(* ========================================================= *)
(*     FB: HLI_CNCChannel                                    *)
(* --------------------------------------------------------- *)
(*   Desc:                                                   *)
(*   Author: MK ,MiB, TV, Rch                                *)
(*   Date: 2020.07.27                                        *)
(*   Rev.: 1.20                                               *)
(*         1.2 Before "start" the state is swicthed to 		 *)
(*				"Selected" and "Ready" to ensure that the    *)	
(*				actual selected program will start 			 *)
(*		   	1.3  BugFix : nChanNo at HLI3_ChannelModeMDI()    *)
(*         	1.4  Implement state switch to "selected" and "ready"  *)         
(*		   	1.5  Channel reset via commanding state 			 *)
(*              RESETTING directly							 *)  
(*		   	1.6  Optimized Channel reset via commanding state *)
(*				RESETTING directly						     *)
(*		   	1.7  Init Paramerer for Manual mode as input parameter*)
(*		   	1.8  BugFix : max index for HLI3_AxisReset		*)
(*		   	1.9  Implementation of HLI3_ManualModeHandler	*)
(*		   	1.10 Implementation of Input bM30Acknowledgement	*)
(*		   	1.12 Optimized Operating modes					*)
(*		   	1.13 Optimized Operating modes				    *)
(*		   	1.14 Optimized M and H Function during Reset     *)
(*		   	1.15 Implementation of ST_CNC_CH_Options Structure *)
(*		   	1.16 BugFix: bCmdReset in mode "Standby" now working *)
(*			1.17 Implementation of CNC PLC Watchdog			*)  
(*			1.18 Optimized CNC PLC Watchdog					*)
(*			1.18 Optimized G201 ManualMode					*)
(*			1.19 Add CmdStandby 							*)
(*			1.20 New Manual Mode 							*)
(* =========================================================*)

IF NOT HLI3_CheckChannelValid(nChannel := nChanIdx) THEN
	RETURN;
END_IF

// CNC PLC Watchdog	
IF NOT stOptions.bDisableCNCPLCWatchDog THEN
	HLI3_SetPLCAlive(nChanIdx :=  nChanIdx);
END_IF

(* handle reset request *)
fbRTrigReset
	(CLK := bStateReset);
	
IF fbRTrigReset.Q THEN
	nStateAutoMDIStart := 0;
	CNCSystem.Channel[nChanIdx].ToolData.bOldToolDataExist := FALSE;
	CNCSystem.Channel[nChanIdx].ToolData.bToolRequest := FALSE;
	CNCSystem.Channel[nChanIdx].ToolData.bResetToolRequest := TRUE;
END_IF

fbRTrigCmdAutomatic(CLK:=bCmdAutomatic);
fbRTrigCmdManual(CLK:=bCmdManual);
fbRTrigCmdReference(CLK:=bCmdReference);
fbRTrigCmdMDI(CLK:=bCmdMDI);
fbRTrigCmdStandby(CLK:=bCmdStandby);	

fbRTrigCmdStart(CLK:=bCmdStart);  
fbRTrigCmdStop(CLK:=bCmdStop);
fbRTrigCmdReset(CLK:=bCmdReset);

(* ************************************* *)
(*  Motion-Control                       *)
(* ************************************* *)

(* EmergencyStop *)
HLI3_ChannelSetEmergencyStop(nChanIdx:=nChanIdx, bEStop := bEmergencyStop);
 
(* Feed Override [0.1%] *)
HLI3_SetChannelOverride(nChanIdx:=nChanIdx, nOverride := nFeedOverride);

(* Rapid feed override [0.1%], must be activated with parameter P-CHAN-00181 *)
HLI3_SetChannelRapidOverride(nChanIdx:=nChanIdx, nOverride := nRapidFeedOverride);

(* Backward Motion *)
HLI3_ChannelSetBackwardMotion(nChanIdx:=nChanIdx, bBackwardMotion:=bBackwardMotion);

(* Program Block Ignore *)
HLI3_ChannelSetProgramBlockIgnore(nChanIdx:=nChanIdx, bPrgBlockIgnore:=bPrgBlockIgnore);

(* Feed Hold *)
HLI3_ChannelSetFeedHold(nChanIdx:=nChanIdx, bFeedHold:=bFeedHold);

(* Single Step *)
HLI3_ChannelSetSingleBlock(nChanIdx:=nChanIdx, bSingleBlock:=bSingleBlock);

(* Reduced Feed *)
HLI3_ChannelSetReducedFeed(nChanIdx:=nChanIdx, bReducedFeed:=bReducedFeed);

(* Syntax Check *)
gpCh[nChanIdx]^.decoder_mc_control.execution_mode.command_w := nSyntaxCheck;

(* Optional stop M01 *)
gpCh[nChanIdx]^.bahn_mc_control.m01_stop_enable.command_w := bM01Stop;

(* ************************************ *)
(*  MHT-Function                        *)
(* ************************************ *)

(* MHT-Function, channel *)
IF NOT stOptions.bDisableMFunctHandling THEN
	ChannelMHTFunction(nChanIdx:=nChanIdx, bM30Acknowledgement := bM30Acknowledgement);
END_IF

(* ************************************* *)
(*  Channel Status Info and error        *)
(* ************************************* *)
HLI3_GetChannelStatusInfo(nChanIdx:=nChanIdx);
HLI3_GetChannelError(nChanIdx:=nChanIdx);

(* ************************************* *)
(*  do single stepping                   *)
(* ************************************* *)
(* Achtung: hier noch anpassen, nur in Abhaengigkeit vom aktuellen Status den Start setzen *)
IF bDoSingleBlock THEN
	bDoSingleBlock := FALSE;
	bStateStart 	:= TRUE;
END_IF

(* ************************************* *)
(*  Operation Modes                      *)
(* ************************************* *)
(* Target modes and states *)
pChannel := ADR(CNCSystem.Channel[nChanIdx]);
OpModes();

(* OperationMode Standby *)
IF stCmdModesStates.stModes.Standby = TRUE THEN
	HLI3_ChannelModeStandby(nChanIdx := nChanIdx,ProgramName:=sProgramName, stCmdModesStates:=stCmdModesStates);
END_IF

(* OperationMode Auto *)
IF stCmdModesStates.stModes.Auto = TRUE THEN
	HLI3_ChannelModeAuto(nChanIdx := nChanIdx, ProgramName:=sProgramName, stCmdModesStates:=stCmdModesStates );
END_IF

(* OperationMode MDI *)
IF stCmdModesStates.stModes.MDI THEN
	(*sProgramName := PLCCncMDIString;*)
	HLI3_ChannelModeMDI(nChanIdx := nChanIdx, pMDIString:=ADR(sMDIString),stCmdModesStates:=stCmdModesStates);
END_IF

(* OperationMode Reference *)
IF stCmdModesStates.stModes.Homing THEN
	sProgramName := '';	(* we choose the default program: rpf.nc *)
	HLI3_ChannelModeReference(nChanIdx := nChanIdx, sRefPosString:=sProgramName, stCmdModesStates:=stCmdModesStates);
END_IF

(* OperationMode Manual *)
(*
IF stCmdModesStates.stModes.Manual THEN	
	HLI3_ChannelModeManual(nChanIdx := nChanIdx, stCmdModesStates:=stCmdModesStates);
END_IF
*)

ModeManual
	(stManualModeParameter  	 	 := stManualModeParameter,
	 stManualModeControlElements	 := stManualModeControlElements,
	 stManualModeControlElementState := stManualModeControlElementState,
	 stCmdModesStates				 := stCmdModesStates,  	
	 arrAxisInG201 				      => stManualModeState[nChanIdx].arrAxisInG201
);
			
(* Reset *)
HLI3_ChannelReset(nChanIdx:=nChanIdx);							(* channel *)
FOR idx := 0 TO UDINT_TO_INT(gNrAx-1) DO							(* axis *)
	HLI3_AxisReset(nChanNo:=nChanIdx+1, nHliAxisIdx:=idx);
END_FOR

ACTION AutoMDIStart:



CASE nStateAutoMDIStart OF
	0:		;(* IDLE *)
	
	10: (* swicth to selected *)
		stCmdModesStates.stStates.Selected := TRUE;
		nStateAutoMDIStart := nStateAutoMDIStart +10;
		
	20: (* wait for selected *)
		IF (pChannel^.ActState =  HLI_IMCM_PROCESS_SELECTED) THEN
			stCmdModesStates.stStates.Ready := TRUE;
			nStateAutoMDIStart := nStateAutoMDIStart +10;
		END_IF
	30: (* Wait for ready and then start*)
		IF (pChannel^.ActState =  HLI_IMCM_PROCESS_READY) THEN
			stCmdModesStates.stStates.Active := TRUE; 
			nStateAutoMDIStart := 0;
		END_IF
	
END_CASE
END_ACTION

ACTION OpModes:
(*************************************************)
(* Restore internal state at first run           *)
(* after PLC reset                               *)
(*************************************************)

IF bCheckOpModeFirst = FALSE THEN
	bCheckOpModeFirst := TRUE;
	currentMode := HLI3_GetChannelMode(nChanIdx:=nChanIdx);
	IF currentMode = HLI_IMCM_STANDBY_MODE THEN
		stCmdModesStates.stModes.Standby := TRUE;
	END_IF
	IF currentMode = HLI_IMCM_AUTOMATIC_MODE THEN
		stCmdModesStates.stModes.Auto := TRUE;
	END_IF
	IF currentMode = HLI_IMCM_MDI_MODE THEN
		stCmdModesStates.stModes.MDI := TRUE;
	END_IF
	IF currentMode = HLI_IMCM_MANUAL_MODE THEN
		stCmdModesStates.stModes.Manual := TRUE;
	END_IF
	IF currentMode = HLI_IMCM_REFERENCE_MODE THEN		
		stCmdModesStates.stModes.Homing := TRUE;
	END_IF
END_IF


(*************************************************)
(* Operation Modes                               *)
(*************************************************)

IF bModeStandby OR fbRTrigCmdStandby.Q THEN
	bModeStandby := FALSE;
	stCmdModesStates.stModes.Standby		:= TRUE;
	stCmdModesStates.stModes.Auto			:= FALSE;
	stCmdModesStates.stModes.MDI			:= FALSE;
	stCmdModesStates.stModes.Manual		:= FALSE;
	stCmdModesStates.stModes.Homing		:= FALSE;
	stCmdModesStates.stStates.Selected	:= TRUE;
END_IF

IF bModeAutomatic OR fbRTrigCmdAutomatic.Q THEN
	bModeAutomatic 				:= FALSE;
	bGoToActive					:= FALSE;
	stCmdModesStates.stModes.Standby		:= FALSE;
	stCmdModesStates.stModes.Auto			:= TRUE;
	stCmdModesStates.stModes.MDI			:= FALSE;
	stCmdModesStates.stModes.Manual		:= FALSE;
	stCmdModesStates.stModes.Homing		:= FALSE;

	stCmdModesStates.stStates.Selected	:= TRUE;
END_IF

IF bModeMDI OR fbRTrigCmdMDI.Q THEN
	bModeMDI := FALSE;
	bGoToActive					:= FALSE;
	stCmdModesStates.stModes.Standby		:= FALSE;
	stCmdModesStates.stModes.Auto			:= FALSE;
	stCmdModesStates.stModes.MDI			:= TRUE;
	stCmdModesStates.stModes.Manual		:= FALSE;
	stCmdModesStates.stModes.Homing		:= FALSE;

	stCmdModesStates.stStates.Selected	:= TRUE;
END_IF

IF bModeManual OR fbRTrigCmdManual.Q THEN
	bModeManual := FALSE;
	stCmdModesStates.stModes.Standby		:= FALSE;
	stCmdModesStates.stModes.Auto			:= FALSE;
	stCmdModesStates.stModes.MDI			:= FALSE;
	stCmdModesStates.stModes.Manual		:= TRUE;
	stCmdModesStates.stModes.Homing		:= FALSE;

	stCmdModesStates.stStates.Active		:= TRUE;
END_IF

IF bModeReference OR fbRTrigCmdReference.Q THEN
	bModeReference := FALSE;
	bGoToActive					:= FALSE;
	stCmdModesStates.stModes.Standby		:= FALSE;
	stCmdModesStates.stModes.Auto			:= FALSE;
	stCmdModesStates.stModes.MDI			:= FALSE;
	stCmdModesStates.stModes.Manual		:= FALSE;
	stCmdModesStates.stModes.Homing		:= TRUE;
	
	IF stOptions.bReferenceModeStartRequired THEN
		stCmdModesStates.stStates.Selected	:= TRUE;
	ELSE
		stCmdModesStates.stStates.Active	:= TRUE;			
	END_IF	
	
END_IF



(*************************************************)
(* Operation States                              *)
(*************************************************)

currentMode := HLI3_GetChannelMode(nChanIdx:=nChanIdx);
currentState := HLI3_GetChannelState(nChanIdx:=nChanIdx);

CASE currentMode OF
	(*-------------------------------------------------------------------*)
	HLI_IMCM_STANDBY_MODE:
		IF bStateReset OR fbRTrigCmdReset.Q THEN
			stCmdModesStates.stModes.Standby := TRUE;
			stCmdModesStates.stStates.Reset := TRUE;
			CNCSystem.Channel[nChanIdx].ToolData.bOldToolDataExist := FALSE;
			CNCSystem.Channel[nChanIdx].ToolData.bToolRequest := FALSE;
			CNCSystem.Channel[nChanIdx].ToolData.bResetToolRequest := TRUE;		
		END_IF

	(*-------------------------------------------------------------------*)
	HLI_IMCM_AUTOMATIC_MODE:
		IF bStateStart OR fbRTrigCmdStart.Q THEN  (* replaced a simple 'start' by a sequence which switches the state to selected and ready*)
			IF currentState <> HLI_IMCM_PROCESS_HOLD AND currentState <> HLI_IMCM_PROCESS_ACTIVE THEN
				nStateAutoMDIStart := 10;
			ELSE
				stCmdModesStates.stStates.Active := TRUE; 
			END_IF					   	
		END_IF
		IF nStateAutoMDIStart <> 0 THEN
			AutoMDIStart();
		END_IF

		IF (bStateStop OR fbRTrigCmdStop.Q) AND currentState <> HLI_IMCM_PROCESS_DESELECTED THEN
			stCmdModesStates.stStates.Hold := TRUE;
		END_IF

		IF bStateReady THEN
			stCmdModesStates.stStates.Ready := TRUE;
		END_IF

		IF bStateReset OR fbRTrigCmdReset.Q THEN
			stCmdModesStates.stStates.Reset := TRUE;
			CNCSystem.Channel[nChanIdx].ToolData.bOldToolDataExist := FALSE;
			CNCSystem.Channel[nChanIdx].ToolData.bToolRequest := FALSE;
			CNCSystem.Channel[nChanIdx].ToolData.bResetToolRequest := TRUE;			
		END_IF
		
		IF bStateSelect THEN
			stCmdModesStates.stStates.Selected := TRUE;
		END_IF		

	(*-------------------------------------------------------------------*)
	HLI_IMCM_MDI_MODE:
		IF bStateStart OR fbRTrigCmdStart.Q THEN
			IF currentState <> HLI_IMCM_PROCESS_HOLD AND currentState <> HLI_IMCM_PROCESS_ACTIVE THEN
				nStateAutoMDIStart := 10;
			ELSE
				stCmdModesStates.stStates.Active := TRUE; 
			END_IF
		END_IF
		
		IF nStateAutoMDIStart <> 0 THEN
			AutoMDIStart();
		END_IF
		
		IF (bStateStop OR fbRTrigCmdStop.Q) AND currentState <> HLI_IMCM_PROCESS_DESELECTED THEN
			stCmdModesStates.stStates.Hold := TRUE;
		END_IF

		IF bStateSelect THEN
			stCmdModesStates.stStates.Selected := TRUE;
		END_IF
		
		IF bStateReady THEN
			stCmdModesStates.stStates.Ready := TRUE;
		END_IF

		IF bStateReset OR fbRTrigCmdReset.Q THEN
			stCmdModesStates.stStates.Reset := TRUE;
			CNCSystem.Channel[nChanIdx].ToolData.bOldToolDataExist := FALSE;
			CNCSystem.Channel[nChanIdx].ToolData.bToolRequest := FALSE;
			CNCSystem.Channel[nChanIdx].ToolData.bResetToolRequest := TRUE;			
		END_IF

	(*-------------------------------------------------------------------*)
	HLI_IMCM_MANUAL_MODE:
		IF bStateStart OR fbRTrigCmdStart.Q OR ((currentState = HLI_IMCM_PROCESS_SELECTED) AND bGoToActive) THEN
			bGoToActive := FALSE;	
			stCmdModesStates.stStates.Active 	:= TRUE;
		END_IF

		IF bStateReady THEN
			stCmdModesStates.stStates.Ready 	:= TRUE;
		END_IF

		IF bStateSelect THEN
			stCmdModesStates.stStates.Selected := TRUE;
		END_IF

		IF bStateStop OR fbRTrigCmdStop.Q THEN
			stCmdModesStates.stStates.Hold := TRUE;
		END_IF

		IF (bStateReset OR fbRTrigCmdReset.Q) THEN	
			CNCSystem.Channel[nChanIdx].ToolData.bOldToolDataExist := FALSE;
			CNCSystem.Channel[nChanIdx].ToolData.bToolRequest := FALSE;
			CNCSystem.Channel[nChanIdx].ToolData.bResetToolRequest := TRUE;
			
			stCmdModesStates.stStates.Reset := TRUE;
			IF stCmdModesStates.stModes.Manual THEN
				bGoToActive := TRUE;
			END_IF
		END_IF

	(*-------------------------------------------------------------------*)
	HLI_IMCM_REFERENCE_MODE:
		IF bStateStart OR fbRTrigCmdStart.Q THEN
			stCmdModesStates.stStates.Active := TRUE;
		END_IF

		IF bStateStop OR fbRTrigCmdStop.Q THEN
			stCmdModesStates.stStates.Hold := TRUE;
		END_IF

		IF bStateReset OR fbRTrigCmdReset.Q THEN
			CNCSystem.Channel[nChanIdx].ToolData.bOldToolDataExist := FALSE;
			CNCSystem.Channel[nChanIdx].ToolData.bToolRequest := FALSE;
			CNCSystem.Channel[nChanIdx].ToolData.bResetToolRequest := TRUE;			
			stCmdModesStates.stStates.Reset := TRUE;
		END_IF
END_CASE


bStateStart 	:= FALSE;
bStateStop 		:= FALSE;
bStateReset 	:= FALSE;
bStateSelect 	:= FALSE;
bStateready 	:= FALSE;
END_ACTION

END_FUNCTION_BLOCK

// CNC/8 Mis/HLI3_SetPLCAlive
FUNCTION HLI3_SetPLCAlive : BOOL
VAR_INPUT
	nChanIdx: INT;		
END_VAR

VAR
	nWatchdogCycles 	: UDINT :=2;	 	
END_VAR

(*
Display PLC is just alive (Trigger Watchdog to MC)
If PLC is stopped here, alive sign is missing.
-> CNC raises error message
-> CNC stoppes movement with internal FEEDHOLD
-> system has to be restarted (after removal of error)
*)

HLI3_SetPLCAlive := FALSE;
IF NOT HLI3_CheckChannelValid(nChannel := nChanIdx) THEN
	RETURN;
END_IF

nWatchdogCycles := 2;

gpCh[nChanIdx]^.head.mc_watchdog.cycle_time_w := CNCSystem.nPLCCycleTime * nWatchdogCycles;   // Watchdog time : PLC Cycle Time * nWatchdogCycles
gpCh[nChanIdx]^.head.mc_watchdog.enable_w := TRUE;
gpCh[nChanIdx]^.head.mc_watchdog.alive_rw := TRUE;

HLI3_SetPLCAlive := TRUE;

END_FUNCTION

// CNC/3 Control/HLI3_ChannelSetEmergencyStop
FUNCTION HLI3_ChannelSetEmergencyStop : BOOL
VAR_INPUT
	/// Number of channel 
	nChanIdx: INT;
	bEStop: BOOL;
END_VAR

(****************************************************************************************)
(* POU:			HLI_ChannelSetEmergenyStop												*)
(* Type:		Function block															*)
(* Customer:	Common																	*)
(* Date:		09/03/12																*)
(* Last:		20/11/12																*)
(* ------------------------------------------------------------------------------------ *)
(* Revision:	1.0																		*)
(* Author:		HR,MiB																	*)
(* Description: (Re-)Sets the channel specific emergency stop unit.						*)
(****************************************************************************************)

HLI3_ChannelSetEmergencyStop := FALSE;
IF NOT HLI3_CheckChannelValid(nChannel := nChanIdx) THEN
	RETURN;
END_IF

(* if the stop button from the HMI is selected the request is set *)
gpCh[nChanIdx]^.bahn_mc_control.emergency_stop.command_w := bEStop;

HLI3_ChannelSetEmergencyStop		:= TRUE;

END_FUNCTION

// CNC/3 Control/HLI3_SetChannelOverride
FUNCTION HLI3_SetChannelOverride : BOOL
VAR_INPUT
	/// Number of channel 
	nChanIdx: INT;
	nOverride: UINT;
END_VAR

(* ========================================================= *)
(*    FUN: HLI_SetChannelOverride                            *)
(* --------------------------------------------------------- *)
(*   Desc: Set the channel Override                          *)
(* Author: MK, MiB                                           *)
(*   Date: 20.11.2012                                        *)
(*   Rev.: 1.2  2017.10.25                                   *)
(* ========================================================= *)

IF NOT HLI3_CheckChannelValid(nChannel := nChanIdx) THEN
	HLI3_SetChannelOverride := FALSE;
	RETURN;
END_IF

(* Limit the override *)
IF nOverride > 2000 THEN nOverride := 2000; END_IF  // MiB 2017.10.25 valid maximum in cnc core is 2000
IF nOverride < 0 THEN nOverride := 0; END_IF

gpCh[nChanIdx]^.bahn_mc_control.override_feedrate.command_w := nOverride;

HLI3_SetChannelOverride := TRUE;

END_FUNCTION

// CNC/3 Control/HLI3_SetChannelRapidOverride
FUNCTION HLI3_SetChannelRapidOverride : BOOL
VAR_INPUT
	/// Number of channel 
	nChanIdx: INT;
	nOverride: UINT;
END_VAR

(* ========================================================= *)
(*    FUN: HLI_SetChannelRapidOverride                       *)
(* --------------------------------------------------------- *)
(*   Desc: Set the channel Override for rapid movements      *)
(*   Author: TV , MiB                                        *)
(*   Date: 07.02.2017                                        *)
(*   Rev.: 1.1                                               *)
(* ========================================================= *)

IF NOT HLI3_CheckChannelValid(nChannel := nChanIdx) THEN
	HLI3_SetChannelRapidOverride := FALSE;
	RETURN;
END_IF

(* Limit the override *)
IF nOverride > 1000	THEN nOverride := 1000; END_IF  // MiB 2017.10.25 maximum is 1000 (ref HLI manual)
IF nOverride < 0 THEN nOverride := 0; END_IF

gpCh[nChanIdx]^.bahn_mc_control.override_rapid_move.enable_w := TRUE;
gpCh[nChanIdx]^.bahn_mc_control.override_rapid_move.command_w := nOverride;

HLI3_SetChannelRapidOverride := TRUE;

END_FUNCTION

// CNC/3 Control/HLI3_ChannelSetBackwardMotion
FUNCTION HLI3_ChannelSetBackwardMotion : BOOL
VAR_INPUT
	/// Number of channel 
	nChanIdx: INT;
	bBackwardMotion: BOOL;
END_VAR

(* ========================================================= *)
(*    FUN: HLI_ChannelSetBackwardMotion                      *)
(* --------------------------------------------------------- *)
(*   Desc:                                                   *)
(* Author: MK, MiB                                           *)
(*   Date: 20.11.2012                                        *)
(*   Rev.: 1.1                                               *)
(* ========================================================= *)

HLI3_ChannelSetBackwardMotion := FALSE;
IF NOT HLI3_CheckChannelValid(nChannel := nChanIdx) THEN
	RETURN;
END_IF

gpCh[nChanIdx]^.bahn_mc_control.backward_motion.command_w := bBackwardMotion;

HLI3_ChannelSetBackwardMotion := TRUE;

END_FUNCTION

// CNC/3 Control/HLI3_ChannelSetProgramBlockIgnore
FUNCTION HLI3_ChannelSetProgramBlockIgnore : BOOL
VAR_INPUT
	/// Number of channel 
	nChanIdx: INT;
	bPrgBlockIgnore: BOOL;
END_VAR

(* ========================================================= *)
(*    FUN: HLI_SetProgramBlockIgnore                         *)
(* --------------------------------------------------------- *)
(*   Desc:                                                   *)
(* Author: MK, MiB , TV                                      *)
(*   Date: 20.12.2012                                        *)
(*   Last: 19.11.2013                                        *)
(*   Rev.: 1.0                                               *)
(* ========================================================= *)

HLI3_ChannelSetProgramBlockIgnore := FALSE;
IF NOT HLI3_CheckChannelValid(nChannel := nChanIdx) THEN
	RETURN;
END_IF

(* program block ignore *)
IF bPrgBlockIgnore THEN
	gpCh[nChanIdx]^.decoder_mc_control.program_block_ignore.command_w := 1;
ELSE
	gpCh[nChanIdx]^.decoder_mc_control.program_block_ignore.command_w := 0;
END_IF

HLI3_ChannelSetProgramBlockIgnore := TRUE;

END_FUNCTION

// CNC/3 Control/HLI3_ChannelSetFeedHold
FUNCTION HLI3_ChannelSetFeedHold : BOOL
VAR_INPUT
	/// Number of channel 
	nChanIdx: INT;
	bFeedHold: BOOL;
END_VAR

(* ========================================================= *)
(*    FUN: HLI_ChannelSetFeedHold                            *)
(* --------------------------------------------------------- *)
(*   Desc:                                                   *)
(* Author: MK , MiB                                          *)
(*   Date: 20.11.2012                                        *)
(*   Rev.: 1.1                                               *)
(* ========================================================= *)

HLI3_ChannelSetFeedHold := FALSE;
IF NOT HLI3_CheckChannelValid(nChannel := nChanIdx) THEN
	RETURN;
END_IF

(* if the stop button from the HMI is selected the request is set *)
gpCh[nChanIdx]^.bahn_mc_control.feedhold.command_w := bFeedHold OR gpCh[nChanIdx]^.bahn_mc_control.feedhold.request_r;
HLI3_ChannelSetFeedHold := TRUE;

END_FUNCTION

// CNC/3 Control/HLI3_ChannelSetSingleBlock
FUNCTION HLI3_ChannelSetSingleBlock : BOOL
VAR_INPUT
	/// Number of channel 
	nChanIdx: INT;
	bSingleBlock: BOOL;
END_VAR

(* ========================================================= *)
(*    FUN: HLI3_ChannelSetSingleBlock                        *)
(* --------------------------------------------------------- *)
(*   Desc:                                                   *)
(* Author: MK ,MiB                                           *)
(*   Date: 20.11.2012                                        *)
(*   Rev.: 1.1                                               *)
(* ========================================================= *)

HLI3_ChannelSetSingleBlock := FALSE;
IF NOT HLI3_CheckChannelValid(nChannel := nChanIdx) THEN
	RETURN;
END_IF
gpCh[nChanIdx]^.bahn_mc_control.single_block.command_w   := bSingleBlock;

HLI3_ChannelSetSingleBlock := TRUE;

END_FUNCTION

// CNC/3 Control/HLI3_ChannelSetReducedFeed
FUNCTION HLI3_ChannelSetReducedFeed : BOOL
VAR_INPUT
	/// Number of channel 
	nChanIdx: INT;
	bReducedFeed: BOOL;
END_VAR

(* ========================================================= *)
(*    FUN: HLI_ChannelSetReducedFeed                         *)
(* --------------------------------------------------------- *)
(*   Desc:                                                   *)
(* Author: MK,MiB                                            *)
(*   Date: 20.11.2012                                        *)
(*   Rev.: 1.1                                               *)
(* ========================================================= *)


HLI3_ChannelSetReducedFeed := FALSE;
IF NOT HLI3_CheckChannelValid(nChannel := nChanIdx) THEN
	RETURN;
END_IF
gpCh[nChanIdx]^.bahn_mc_control.reduced_speed.command_w := bReducedFeed;
HLI3_ChannelSetReducedFeed := TRUE;

END_FUNCTION

// CNC/3 Control/HLI3_GetChannelStatusInfo
FUNCTION HLI3_GetChannelStatusInfo : BOOL
VAR_INPUT
	/// Number of channel 
	nChanIdx: INT;
END_VAR
VAR
	pChannel: POINTER TO ST_CNCChannel;
END_VAR

(* ========================================================= *)
(*    FUN: HLI_GetStatusInfo                                 *)
(* --------------------------------------------------------- *)
(*   Desc: Status Info from the HLI Interface                *)
(* Author: MK,Mib                                            *)
(*   Date: 18.07.2002                                        *)
(*   Rev.: 1.0                                               *)
(* ========================================================= *)

IF NOT HLI3_CheckChannelValid(nChannel := nChanIdx) THEN
	RETURN;
END_IF


pChannel := ADR(CNCSystem.Channel[nChanIdx]);
pChannel^.ActMode := HLI3_GetChannelMode(nChanIdx:=nChanIdx);
pChannel^.ActState := HLI3_GetChannelState(nChanIdx:=nChanIdx);

pChannel^.Mode.Standby := FALSE;
pChannel^.Mode.Auto := FALSE;
pChannel^.Mode.Homing := FALSE;
pChannel^.Mode.MDI := FALSE;
pChannel^.Mode.Manual := FALSE;

(* Translate mode *)
CASE pChannel^.ActMode OF
	HLI_IMCM_MODE:					pChannel^.ActModeString := 'Mode';
	HLI_IMCM_STANDBY_MODE:			pChannel^.ActModeString := 'StandbyMode'; pChannel^.Mode.Standby:=TRUE;
	HLI_IMCM_AUTOMATIC_MODE:		pChannel^.ActModeString := 'AutomaticMode'; pChannel^.Mode.Auto:=TRUE;
	HLI_IMCM_MDI_MODE:				pChannel^.ActModeString := 'MDIMode'; pChannel^.Mode.MDI:=TRUE;
	HLI_IMCM_MANUAL_MODE:			pChannel^.ActModeString := 'ManualMode'; pChannel^.Mode.Manual:=TRUE;;
	HLI_IMCM_REFERENCE_MODE:		pChannel^.ActModeString := 'ReferenceMode'; pChannel^.Mode.Homing:=TRUE;
ELSE
	pChannel^.ActModeString := '---';
END_CASE;

pChannel^.State.Selected:=FALSE;
pChannel^.State.Ready:=FALSE;
pChannel^.State.Active:=FALSE;
pChannel^.State.Hold:=FALSE;
pChannel^.State.Error:=FALSE;

(* Translate state *)
CASE pChannel^.ActState OF
	HLI_IMCM_PROCESS_DESELECTED:	pChannel^.ActStateString := 'Deselected';
	HLI_IMCM_PROCESS_SELECTED:		pChannel^.ActStateString := 'Selected'; pChannel^.State.Selected:=TRUE;
	HLI_IMCM_PROCESS_READY:			pChannel^.ActStateString := 'Ready'; pChannel^.State.Ready:=TRUE;
	HLI_IMCM_PROCESS_ACTIVE:		pChannel^.ActStateString := 'Active'; pChannel^.State.Active:=TRUE;
	HLI_IMCM_PROCESS_HOLD:			pChannel^.ActStateString := 'Hold'; pChannel^.State.Hold:=TRUE;
	HLI_IMCM_PROCESS_ERROR:			pChannel^.ActStateString := 'Error'; pChannel^.State.Error:=TRUE;
	HLI_IMCM_PROCESS_SELECTING:		pChannel^.ActStateString := 'Selecting';
	HLI_IMCM_PROCESS_DESELECTING:	pChannel^.ActStateString := 'Deselecting';
	HLI_IMCM_PROCESS_PREPARING:		pChannel^.ActStateString := 'Preparing';
	HLI_IMCM_PROCESS_CLEARING:		pChannel^.ActStateString := 'Clearing';
	HLI_IMCM_PROCESS_STARTING:		pChannel^.ActStateString := 'Starting';
	HLI_IMCM_PROCESS_ABORTING:		pChannel^.ActStateString := 'Aborting';
	HLI_IMCM_PROCESS_STOPPING:		pChannel^.ActStateString := 'Stopping';
	HLI_IMCM_PROCESS_RESUMING:		pChannel^.ActStateString := 'Resuming';
	HLI_IMCM_PROCESS_RESETTING:		pChannel^.ActStateString := 'Resetting';
	HLI_IMCM_PROCESS_FINISHING:		pChannel^.ActStateString := 'Finishing';
ELSE
	pChannel^.ActStateString := '---';
END_CASE;

END_FUNCTION

// CNC/3 Control/HLI3_GetChannelMode
FUNCTION HLI3_GetChannelMode : UDINT
VAR_INPUT
	/// Number of channel 
	nChanIdx: INT;
END_VAR

(* ========================================================= *)
(*    FUN: HLI_GetChannelMode                                *)
(* --------------------------------------------------------- *)
(*   Desc:                                                   *)
(* Author: MK                                                *)
(*   Date: 18.07.2002                                        *)
(*   Rev.: 1.0                                               *)
(* ========================================================= *)
HLI3_GetChannelMode := 0;
IF NOT HLI3_CheckChannelValid(nChannel := nChanIdx) THEN
	RETURN;
END_IF

(* if the stop button from the HMI is selected the request is set *)
HLI3_GetChannelMode := gpCh[nChanIdx]^.channel_mc_control.mode_and_state.state_r.mode;

END_FUNCTION

// CNC/3 Control/HLI3_GetChannelState
FUNCTION HLI3_GetChannelState : UDINT
VAR_INPUT
	/// Number of channel 
	nChanIdx: INT;
END_VAR

(* ========================================================= *)
(*    FUN: HLI3_GetChannelState                              *)
(* --------------------------------------------------------- *)
(*   Desc:                                                   *)
(* Author: MK                                                *)
(*   Date: 18.07.2002                                        *)
(*   Rev.: 1.0                                               *)
(* ========================================================= *)

HLI3_GetChannelState := 0;
IF NOT HLI3_CheckChannelValid(nChannel := nChanIdx) THEN
	RETURN;
END_IF

(* if the stop button from the HMI is selected the request is set *)
HLI3_GetChannelState := gpCh[nChanIdx]^.channel_mc_control.mode_and_state.state_r.state;

END_FUNCTION

// CNC/3 Control/HLI3_GetChannelError
FUNCTION HLI3_GetChannelError : BOOL
VAR_INPUT
	/// Number of channel 
	nChanIdx: INT;
END_VAR
VAR
	pChannel: POINTER TO ST_CNCChannel;
END_VAR

(* ========================================================= *)
(*    FUN: HLI_GetChannelError                               *)
(* --------------------------------------------------------- *)
(*   Desc: Gets the channel error                            *)
(* Return: The error flag of the channel                     *)
(* Author: MK , MiB, TV                                      *)
(*   Date: 08.07.2015                                        *)
(*   Rev.: 1.3                                               *)
(* ========================================================= *)

IF NOT HLI3_CheckChannelValid(nChannel := nChanIdx) THEN
	RETURN;
END_IF

pChannel := ADR(CNCSystem.Channel[nChanIdx]);

(* Visualisation of Mode and State *)
pChannel^.ActMode  := HLI3_GetChannelMode(nChanIdx:=nChanIdx);
pChannel^.ActState := HLI3_GetChannelState(nChanIdx:=nChanIdx);

(* Error messages id *)
IF pChannel^.ActState = HLI_IMCM_PROCESS_ERROR THEN
	pChannel^.Error := TRUE;	
ELSE
	pChannel^.Error := FALSE;	
END_IF

END_FUNCTION

// CNC/4 MHT-Function/HLI3_QuitChannelMHTFunction
FUNCTION_BLOCK HLI3_QuitChannelMHTFunction
VAR_INPUT
	/// Number of channel 
	nChanIdx: INT;
	bM30Acknowledgement : BOOL;
END_VAR
VAR_OUTPUT
	bOK: BOOL;
END_VAR
VAR
	ChannelMFunction: HLI3_DoChannelMFunction;
	ChannelTFunction: HLI3_DoChannelTFunction;
	ChannelHFunction: HLI3_DoChannelHFunction;
	/// local pointer to Data of actual Channel 
	pChannelData: POINTER TO HIGH_LEVEL_INTERFACE_CH;
	/// local pointer to actual techno unit 
	pActTechnoUnit: POINTER TO TECHNO_UNIT_CH;
	/// Index of axis specific technology function at HLI 
	nTechFctMaxIdx: UINT;
	nTechFctAnzahl : UINT; 
	/// loop variable 
	idx: UINT;
	/// number of M-function 
	nFuncNr: UDINT;
	nArgument: DINT;
	/// basis id of a tool 
	nToolBasicId: UDINT;
	pMHProcess: POINTER TO HLI_M_H_PROZESS;
	pSProcess: POINTER TO HLI_S_PROZESS;
	pTProcess: POINTER TO HLI_T_PROZESS;
	stAttributeData: St_TechnoAttributeData;	
END_VAR

(* ========================================================= *)
(*     FB: HLI3_QuitChannelMHTFunction                        *)
(* --------------------------------------------------------- *)
(*   Desc:                                                   *)
(* Author: MK                                                *)
(*   Rev.: 1.1                                               *)
(*   Date: 18.07.2002                                        *)
(*       : 08.04.2005                                        *)
(*          24.11.2010 MiB Erweiterung um H Funktionen 		 *)
(* ========================================================= *)
(* Rev.:	1.2												 *)
(* Date:	02.10.2010                                    	 *)
(* Author:	HR												 *)
(* Author:	Added support for additional m function number	 *)
(* ========================================================= *)
(* Rev.:	1.3												 *)
(* Date:	26.01.2011                                    	 *)
(* Author:	HR												 *)
(* Author:	Added support for additional h function number	 *)
(* ========================================================= *)
(* Rev.:	1.4												 *)
(* Date:	20.11.2012                                    	 *)
(* Author:	MiB												 *)
(* Author:	TC3												 *)
(* ========================================================= *)
(* Rev.:	1.4.1									         *)
(* Date:	15.07.2013                                    	 *)
(* Author:	TV												 *)
(* ========================================================= *)
(* Rev.:	1.4.2									         *)
(* Date:	22.09.2016                                    	 *)
(* Author:	TV												 *)
(* ========================================================= *)
(* ========================================================= *)
(* Rev.:	1.4.3									         *)
(* Date:	01.12.2017                                    	 *)
(* Author:	TV												 *)
(*													 	 	 *)
(* ========================================================= *)

IF NOT HLI3_CheckChannelValid(nChannel := nChanIdx) THEN
	bOK := FALSE;
	RETURN; (* A b b r u c h *)
END_IF


(* get pointer to channel data *)
pChannelData := gpCh[nChanIdx];

pActTechnoUnit := ADR(pChannelData^.techno_unit_std_sync[0]);

(* test if there are open synchronisations  *)
IF pChannelData^.used_units_std_sync_r > 0 THEN

	nTechFctAnzahl := pChannelData^.used_units_std_sync_r;
	
	IF nTechFctAnzahl  > 0 THEN

        nTechFctMaxIdx := nTechFctAnzahl  - 1;  

		FOR idx := 0 TO nTechFctMaxIdx DO
			(* get pointer to actual techno unit *)
			pActTechnoUnit := ADR(pChannelData^.techno_unit_std_sync[idx]);
		
		
			(* test if this M-function has to be acknowledged *)
			IF pActTechnoUnit^.please_rw = TRUE AND				(* request from CNC *)
			   pActTechnoUnit^.done_w = FALSE AND				(* not acknowledged *)
			   pActTechnoUnit^.fkt_ctrl_r = HLI_INTF_M_FKT		(* M-function *)
			THEN
				(* Read number of M-function *)
				pMHProcess := ADR(pActTechnoUnit^.attribut_r.data[0]);
				nFuncNr    := pMHProcess^.nr;
				nArgument	:= pMHProcess^.add_nr_r;
				
				
				stAttributeData.nFunctionNumber_r := pMHProcess^.nr;
				stAttributeData.nTime_r		:= pMHProcess^.zeit;
				stAttributeData.nArgument_r 		:= pMHProcess^.add_nr_r;
				stAttributeData.nBlockNumber_r 	:= pMHProcess^.satz_nr;
				stAttributeData.nPrgLineNumber_r	:= pMHProcess^.prg_zeilen_nr;
				
		
				ChannelMFunction(nChanIdx:=nChanIdx, stTechnoAttributeData := stAttributeData, bM30Acknowledgement := bM30Acknowledgement);
				IF ChannelMFunction.bBusy = FALSE THEN
					(* acknowledge this M-function *)
					pActTechnoUnit^.please_rw := FALSE;
					pActTechnoUnit^.done_w := TRUE;				
				END_IF
		
				bOK := TRUE;
			END_IF
	
	
			(* test if this H-function has to be acknowledged *)
			IF pActTechnoUnit^.please_rw = TRUE AND						(* request from CNC *)
			   pActTechnoUnit^.done_w = FALSE AND						(* not acknowledged *)
			   pActTechnoUnit^.fkt_ctrl_r = HLI_INTF_H_FKT		(* H-function *)
			THEN
				(* Read number of H-function *)
				pMHProcess := ADR(pActTechnoUnit^.attribut_r.data[0]);
				stAttributeData.nFunctionNumber_r := pMHProcess^.nr;
				stAttributeData.nTime_r		:= pMHProcess^.zeit;
				stAttributeData.nArgument_r 		:= pMHProcess^.add_nr_r;
				stAttributeData.nBlockNumber_r 	:= pMHProcess^.satz_nr;
				stAttributeData.nPrgLineNumber_r	:= pMHProcess^.prg_zeilen_nr;
		
				ChannelHFunction(nChanIdx:=nChanIdx, stTechnoAttributeData:= stAttributeData);
	
				(* acknowledge this H-function *)
				IF ChannelHFunction.bBusy = FALSE THEN
						(* acknowledge this H-function *)
					pActTechnoUnit^.please_rw := FALSE;
					pActTechnoUnit^.done_w := TRUE;			
				END_IF
				bOK := TRUE;
			END_IF
		
			(* test if this T-function has to be acknowledged *)
			IF pActTechnoUnit^.please_rw = TRUE AND				(* request from CNC *)
			   pActTechnoUnit^.done_w = FALSE AND				(* not acknowledged *)
			   pActTechnoUnit^.fkt_ctrl_r = HLI_INTF_TOOL		(* T-function *)
			THEN
				(* Read number of T-function *)
				pTProcess    := ADR(pActTechnoUnit^.attribut_r.data[0]);
				nToolBasicId := DINT_TO_UDINT(pTProcess^.id.basic);
		
				ChannelTFunction(nChanIdx:=nChanIdx, nFuncNr:=nToolBasicId);
		
				(* acknowledge this T-function *)
				pActTechnoUnit^.please_rw := FALSE;
				pActTechnoUnit^.done_w := TRUE;				
				bOK := TRUE;
			END_IF
		
		END_FOR
	
	END_IF

END_IF


(*
	HLI_INTF_H_FKT                 :    INT:=2;
	HLI_INTF_SPINDEL              :    INT:=3;
	HLI_INTF_TOOL                 :    INT:=4;
	GCW_250_HLIIntfAxBlock              :    INT:=5;
	GCW_250_HLIIntfVEVariable           :    INT:=6;
	GCW_250_HLIIntfVEVariable_1         :    INT:=7;
	GCW_250_HLIIntfVEVariable_2         :    INT:=8;
	GCW_250_HLIIntfUnknown              :    INT:=9;
*)

(*******************************************************************************************************************)

FOR idx := 0 TO INT_TO_UINT(HLI_TU_CH_LATE_SYNC_MAXIDX) DO
	IF pChannelData^.techno_unit_late_sync[idx].please_rw = TRUE
	AND pChannelData^.techno_unit_late_sync[idx].done_w = FALSE THEN

		(* get pointer to actual techno unit *)
		pActTechnoUnit := ADR(pChannelData^.techno_unit_late_sync[idx]);

		IF pActTechnoUnit^.please_rw = TRUE AND				(* request from CNC *)
			pActTechnoUnit^.done_w = FALSE AND				(* not acknowledged *)
			pActTechnoUnit^.fkt_ctrl_r = HLI_INTF_M_FKT		(* M-function *)
		THEN
			pMHProcess := ADR(pActTechnoUnit^.attribut_r.data[0]);
			nFuncNr    := pMHProcess^.nr;
			
			stAttributeData.nFunctionNumber_r := pMHProcess^.nr;
			stAttributeData.nTime_r		:= pMHProcess^.zeit;
			stAttributeData.nArgument_r 		:= pMHProcess^.add_nr_r;
			stAttributeData.nBlockNumber_r 	:= pMHProcess^.satz_nr;
			stAttributeData.nPrgLineNumber_r	:= pMHProcess^.prg_zeilen_nr;

			ChannelMFunction(nChanIdx:=nChanIdx, stTechnoAttributeData:=stAttributeData);
			IF ChannelMFunction.bBusy = FALSE THEN
			(* acknowledge this M-function *)
			pActTechnoUnit^.please_rw := FALSE;
			pActTechnoUnit^.done_w := TRUE;
			
			(* ADSLOGDINT( msgCtrlMask := ADSLOG_MSGTYPE_MSGBOX OR
										ADSLOG_MSGTYPE_LOG,
						msgFmtStr := 'Channel acknowledge of M-function: %d',
						dintArg := pMHProcess^.nr);
			*)
		END_IF
		bOK := TRUE;

	(*	ELSIF   pActTechnoUnit^.fkt_ctrl_r = HLI_INTF_SPINDEL THEN (* spindle-function *)

 			(* Example: read number of S-function *)
			pSProzess := ADR(pActTechnoUnit^.attribut_r.data[0]);
			ADSLOGDINT( msgCtrlMask := ADSLOG_MSGTYPE_MSGBOX OR
										ADSLOG_MSGTYPE_LOG,
						msgFmtStr := 'Late synch : %d',
						dintArg := pSProzess^.move_cmd);

		ELSIF   pActTechnoUnit^.fkt_ctrl_r = HLI_INTF_TOOL THEN

			pHLI_T_PROZESS := ADR(pActTechnoUnit^.attribut_r.data[0]);
			ADSLOGDINT( msgCtrlMask := ADSLOG_MSGTYPE_MSGBOX OR
										ADSLOG_MSGTYPE_LOG,
						msgFmtStr := 'Late tool process: %d',
						dintArg := pTProcess^.id.basic);*)
		(*ELSE
				ADSLOGDINT( msgCtrlMask := ADSLOG_MSGTYPE_MSGBOX OR
											ADSLOG_MSGTYPE_LOG,
							msgFmtStr := 'Channel acknowledge unknown type: %d',
							dintArg := pActTechnoUnit^.fkt_ctrl_r);*)
		END_IF

	END_IF
END_FOR
(**********************************************************************************************************************)

END_FUNCTION_BLOCK

// CNC/4 MHT-Function/HLI3_DoChannelMFunction
FUNCTION_BLOCK HLI3_DoChannelMFunction
VAR_INPUT
	/// Channel number 
	nChanIdx: INT;
	stTechnoAttributeData: St_TechnoAttributeData;
	bM30Acknowledgement : BOOL;
END_VAR
VAR_OUTPUT
	bBusy: BOOL;
END_VAR
VAR
	pChannel: POINTER TO ST_CncChannel;
END_VAR

(* ========================================================= *)
(*     FB: HLI_DoChannelMFunction                            *)
(* --------------------------------------------------------- *)
(*   Desc:                                                   *)
(* Author: MK                                                *)
(*   Rev.: 1.1                                               *)
(*   Date: 18.07.2002                                        *)
(*       : 08.04.2005                                        *)
(* ========================================================= *)
(* Rev.:	1.2												 *)
(* Date:	02.10.2010                                   	 *)
(* Author:	HR												 *)
(* Author:	Added support for additional m function number	 *)
(*			via new input variable 'nArg'				 	 *)
(* ========================================================= *)
(* Rev.:	1.3												 *)
(* Date:	23.11.2012                                   	 *)
(* Author:	TV, MiB											 *)
(* Author:	structure St_TechnoAttributeData instead of      *)
(*			simple bool array	 							 *)
(* ========================================================= *)
(* Rev.:	1.4												 *)
(* Date:	22.09.2016                                   	 *)
(* Author:	TV 											 	 *)
(* Dec:		Implementation of Input bM30Acknowledgement      *)
(*				 							                 *)
(* ========================================================= *)

bBusy := TRUE;
IF NOT HLI3_CheckChannelValid(nChannel := nChanIdx) THEN
	RETURN; (* A b b r u c h *)
END_IF


pChannel := ADR(CNCSystem.Channel[nChanIdx]);

(* Synch M-Functions *)
IF stTechnoAttributeData.nFunctionNumber_r > 0 AND stTechnoAttributeData.nFunctionNumber_r < 1000 THEN
	IF NOT pChannel^.M[stTechnoAttributeData.nFunctionNumber_r].bRes THEN					(* M-Function not set *)
		pChannel^.M[stTechnoAttributeData.nFunctionNumber_r].bState_rw				:= TRUE;	(* set M-Function *)
		pChannel^.M[stTechnoAttributeData.nFunctionNumber_r].nArgument_r		:= stTechnoAttributeData.nArgument_r;
		pChannel^.M[stTechnoAttributeData.nFunctionNumber_r].nBlockNumber_r		:= stTechnoAttributeData.nBlockNumber_r;
		pChannel^.M[stTechnoAttributeData.nFunctionNumber_r].nPrgLineNumber_r	:= stTechnoAttributeData.nPrgLineNumber_r;
		pChannel^.M[stTechnoAttributeData.nFunctionNumber_r].nFunctionNumber_r	:= stTechnoAttributeData.nFunctionNumber_r;
		pChannel^.M[stTechnoAttributeData.nFunctionNumber_r].nTime_r			:= stTechnoAttributeData.nTime_r;		
		pChannel^.M[stTechnoAttributeData.nFunctionNumber_r].bRes 				:= TRUE;	(* set acknowledge *)
		pChannel^.actM_r := CONCAT('M', UDINT_TO_STRING(stTechnoAttributeData.nFunctionNumber_r));
	ELSE
		IF NOT pChannel^.M[stTechnoAttributeData.nFunctionNumber_r].bState_rw THEN				(* wait for quit *)
			pChannel^.M[stTechnoAttributeData.nFunctionNumber_r].bRes 			:= FALSE;	(* quit the ack *)
			pChannel^.M[stTechnoAttributeData.nFunctionNumber_r].nArgument_r	:= 0;		(* reset the argument *)
			pChannel^.M[stTechnoAttributeData.nFunctionNumber_r].nBlockNumber_r		:= 0;
			pChannel^.M[stTechnoAttributeData.nFunctionNumber_r].nPrgLineNumber_r	:= 0;
			pChannel^.M[stTechnoAttributeData.nFunctionNumber_r].nFunctionNumber_r	:= 0;
			pChannel^.M[stTechnoAttributeData.nFunctionNumber_r].nTime_r			:= 0;				
			pChannel^.actM_r :='';
			bBusy 							:= FALSE;	(* quit *)
		END_IF
	END_IF
END_IF


(* Quit M00, M01, M02 , M17, M29, M30 *)
IF 	stTechnoAttributeData.nFunctionNumber_r = 0 OR 
	stTechnoAttributeData.nFunctionNumber_r = 01 OR 
	stTechnoAttributeData.nFunctionNumber_r = 02 OR 
	stTechnoAttributeData.nFunctionNumber_r = 17  OR 
	stTechnoAttributeData.nFunctionNumber_r = 29  OR 
	(stTechnoAttributeData.nFunctionNumber_r = 30 AND bM30Acknowledgement) THEN
		pChannel^.M[stTechnoAttributeData.nFunctionNumber_r].bState_rw 			:= FALSE;
		pChannel^.M[stTechnoAttributeData.nFunctionNumber_r].nArgument_r	:= 0;
		pChannel^.M[stTechnoAttributeData.nFunctionNumber_r].bRes 			:= FALSE;
		bBusy 							:= FALSE;
END_IF

END_FUNCTION_BLOCK

// CNC/4 MHT-Function/HLI3_DoChannelTFunction
FUNCTION_BLOCK HLI3_DoChannelTFunction
VAR_INPUT
	/// Channel number 
	nChanIdx: INT;
	/// Number of T-function 
	nFuncNr: UDINT;
END_VAR
VAR_OUTPUT
	bBusy: BOOL;
END_VAR
VAR
	bStartTimer: BOOL;
END_VAR

(* ========================================================= *)
(*     FB: HLI_DoChannelTFunction                            *)
(* --------------------------------------------------------- *)
(*   Desc:                                                   *)
(* Author: MK, MiB                                           *)
(*   Rev.: 1.1                                               *)
(*   Date: 18.07.2002                                        *)
(*       : 08.04.2005, 03.03.2016 							 *)
(* ========================================================= *)


bBusy := FALSE;
RETURN;

IF NOT HLI3_CheckChannelValid(nChannel := nChanIdx) THEN
	RETURN; (* A b b r u c h *)
END_IF
bBusy := TRUE;

CASE nChanIdx OF
	0:	(* cnc channel 1 -------------------------------------- *)
		CASE nFuncNr OF
			0:		bBusy := FALSE;
			1:		bBusy := FALSE;
			2:		bBusy := FALSE;
			3:		bBusy := FALSE;
			4:		bBusy := FALSE;
			5:		bBusy := FALSE;
			6:		bBusy := FALSE;
			7:		bBusy := FALSE;
			8:		bBusy := FALSE;

			ELSE
			ADSLOGDINT( msgCtrlMask :=    ADSLOG_MSGTYPE_MSGBOX
			                           OR ADSLOG_MSGTYPE_LOG,
						msgFmtStr   := 'T-Funktion (%d), Channel 1, HLI_DoChannelTFunction() not implemented!',
						dintArg     := UDINT_TO_DINT(nFuncNr));
				(* Quit the M-Function *)
				bBusy := TRUE;
		END_CASE;


	1:	(* cnc channel 2 -------------------------------------- *)
		CASE nFuncNr OF
			0:		bBusy := FALSE;
			1:		bBusy := FALSE;
			2:		bBusy := FALSE;
			3:		bBusy := FALSE;


			ELSE
				ADSLOGDINT( msgCtrlMask :=    ADSLOG_MSGTYPE_MSGBOX
				                           OR ADSLOG_MSGTYPE_LOG,
							msgFmtStr   := 'T-Funktion (%d), Channel 2, HLI_DoChannelTFunction() not implemented!',
							dintArg     := UDINT_TO_DINT(nFuncNr));
				(* Quit the M-Function *)
				bBusy := FALSE;
		END_CASE;

ELSE
	ADSLOGDINT( msgCtrlMask :=    ADSLOG_MSGTYPE_MSGBOX
	                           OR ADSLOG_MSGTYPE_LOG,
				msgFmtStr   := 'Unknown channel number (%d) in HLI_DoChannelTFunction',
				dintArg     := INT_TO_DINT(nChanIdx));
	bBusy := FALSE;
END_CASE;

END_FUNCTION_BLOCK

// CNC/4 MHT-Function/HLI3_DoChannelHFunction
FUNCTION_BLOCK HLI3_DoChannelHFunction
VAR_INPUT
	/// Channel number 
	nChanIdx: INT;
	stTechnoAttributeData: St_TechnoAttributeData;
END_VAR
VAR_OUTPUT
	bBusy: BOOL;
END_VAR
VAR
	pChannel: POINTER TO ST_CncChannel;
END_VAR

(* ========================================================= *)
(*     FB: HLI_DoChannelHFunction                            *)
(* --------------------------------------------------------- *)
(*   Desc:                                                   *)
(* Author: MiB                                               *)
(*   Rev.: 1.0                                               *)
(*   Date: 24.11.2010                                        *)
(*       : 08.04.2005                                        *)
(* ========================================================= *)
(* Rev.:	1.2												 *)
(* Date:	26.01.2011                                   	 *)
(* Author:	HR												 *)
(* Author:	Added support for additional h function number	 *)
(*			via new input variable 'nArg'				 	 *)
(* ========================================================= *)
bBusy := TRUE;

IF NOT HLI3_CheckChannelValid(nChannel := nChanIdx) THEN
	RETURN; (* A b b r u c h *)
END_IF


pChannel := ADR(CNCSystem.Channel[nChanIdx]);

(* Synch M-Functions *)
IF stTechnoAttributeData.nFunctionNumber_r > 0 AND stTechnoAttributeData.nFunctionNumber_r < 1000 THEN
	IF NOT pChannel^.H[stTechnoAttributeData.nFunctionNumber_r].bRes THEN					(* M-Function not set *)
		pChannel^.H[stTechnoAttributeData.nFunctionNumber_r].bState_rw				:= TRUE;	(* set M-Function *)
		pChannel^.H[stTechnoAttributeData.nFunctionNumber_r].nArgument_r		:= stTechnoAttributeData.nArgument_r;
		pChannel^.H[stTechnoAttributeData.nFunctionNumber_r].nBlockNumber_r		:= stTechnoAttributeData.nBlockNumber_r;
		pChannel^.H[stTechnoAttributeData.nFunctionNumber_r].nPrgLineNumber_r	:= stTechnoAttributeData.nPrgLineNumber_r;
		pChannel^.H[stTechnoAttributeData.nFunctionNumber_r].nFunctionNumber_r	:= stTechnoAttributeData.nFunctionNumber_r;
		pChannel^.H[stTechnoAttributeData.nFunctionNumber_r].nTime_r			:= stTechnoAttributeData.nTime_r;		
		pChannel^.H[stTechnoAttributeData.nFunctionNumber_r].bRes 				:= TRUE;	(* set acknowledge *)
		pChannel^.actH_r := CONCAT('H', UDINT_TO_STRING(stTechnoAttributeData.nFunctionNumber_r));
	ELSE
		IF NOT pChannel^.H[stTechnoAttributeData.nFunctionNumber_r].bState_rw THEN				(* wait for quit *)
			pChannel^.H[stTechnoAttributeData.nFunctionNumber_r].bRes 			:= FALSE;	(* quit the ack *)
			pChannel^.H[stTechnoAttributeData.nFunctionNumber_r].nArgument_r	:= 0;		(* reset the argument *)
			pChannel^.H[stTechnoAttributeData.nFunctionNumber_r].nBlockNumber_r		:= 0;
			pChannel^.H[stTechnoAttributeData.nFunctionNumber_r].nPrgLineNumber_r	:= 0;
			pChannel^.H[stTechnoAttributeData.nFunctionNumber_r].nFunctionNumber_r	:= 0;
			pChannel^.h[stTechnoAttributeData.nFunctionNumber_r].nTime_r			:= 0;
			pChannel^.actH_r := '';					
			bBusy 							:= FALSE;	(* quit *)
		END_IF
	END_IF
END_IF

END_FUNCTION_BLOCK

// CNC/3 Control/FB_Diag
FUNCTION_BLOCK FB_Diag
VAR_OUTPUT
	Alarm: BOOL;
	Vorwarn: BOOL;
	Meld: BOOL;
END_VAR

Alarm := TRUE;
Vorwarn := TRUE;
Meld := TRUE;

END_FUNCTION_BLOCK

// CNC/3 Control/HLI3_ChannelSetSuspendAxisOutput
FUNCTION HLI3_ChannelSetSuspendAxisOutput : BOOL
VAR_INPUT
	/// Number of channel 
	nChanIdx: INT;
	bSuspendAxis: BOOL;
END_VAR

(* ========================================================= *)
(*    FUN: HLI_ChannelSuspendAxisOutput                      *)
(* --------------------------------------------------------- *)
(*   Desc:                                                   *)
(* Author: MK , MiB                                          *)
(*   Date: 20.11.2012                                        *)
(*   Rev.: 1.1                                               *)
(* ========================================================= *)
HLI3_ChannelSetSuspendAxisOutput := TRUE;
IF NOT HLI3_CheckChannelValid(nChannel := nChanIdx) THEN
	RETURN;
END_IF
gpCh[nChanIdx]^.bahn_mc_control.suspend_axis_output.command_w := bSuspendAxis;
HLI3_ChannelSetSuspendAxisOutput := TRUE;

END_FUNCTION

// CNC/3 Control/HLI3_GetActualAxisPos
FUNCTION HLI3_GetActualAxisPos : LREAL
VAR_INPUT
	///Achs ID
	nHliAxisIdx: INT;
END_VAR
VAR
	HLI_GetActualAxisPos: DINT;
END_VAR



IF NOT (HLI3_CheckAxisValid(nHliAxisIdx := nHliAxisIdx)) THEN
	HLI3_GetActualAxisPos := -1;
	RETURN;
END_IF

HLI3_GetActualAxisPos:=  gpAx[nHliAxisIdx]^.lr_state.current_position_acs_r;

END_FUNCTION

// CNC/3 Control/HLI3_GetAxisReferenceState
FUNCTION HLI3_GetAxisReferenceState : BOOL
VAR_INPUT
	nHliAxisIdx: INT;
END_VAR


IF NOT HLI3_CheckAxisValid(nHliAxisIdx := nHliAxisIdx) THEN
	HLI3_GetAxisReferenceState := FALSE;
	RETURN;
END_IF

HLI3_GetAxisReferenceState:= gpAx[nHliAxisIdx]^.lr_state.homing_done_r;

END_FUNCTION

// CNC/3 Control/HLI3_GetAxisScaling
FUNCTION_BLOCK HLI3_GetAxisScaling
VAR_INPUT
	bExec:		BOOL;	// riding edge to start read
	nHliAxisIdx: INT;	
END_VAR
VAR_OUTPUT
	Scaling	:	LREAL;	// scalingfactor inc/0.1µm
	bBusy: 		BOOL;
	bError: 	BOOL;
	nErrorID: 	UDINT;
END_VAR
VAR
	fbAdsRead: ADSREAD;
END_VAR

(* ========================================================= *)
(*    FUN: HLI3_GetAxisScaling	                   		 	*)
(* --------------------------------------------------------- *)
(*   Desc: Gets the scaling factor of an axis   			 *)
(*															 *)
(* Return: Scaling in INC/0.1µm							 	*)
(* Author: MiB                                               *)
(* Date: 29.08.2019                                        *)
(* Rev.: 1.0                                               *)
(* ========================================================= *)



IF NOT (HLI3_CheckAxisValid(nHliAxisIdx := nHliAxisIdx)) THEN
	Scaling := 0.0;
	bError := TRUE;
	nErrorId := 1000;  // wrong HLI index
	RETURN;
END_IF


fbAdsRead(
	NETID:= '' , 
	PORT:= 551, 
	IDXGRP:= 16#23300 , 
	IDXOFFS:= 16#10000 * (nHliAxisIdx+1) + 16#1 , 
	LEN:= SIZEOF(Scaling) , 
	DESTADDR:= ADR(Scaling),
	READ:= bExec, 
	TMOUT:= , 
	BUSY=> bBusy, 
	ERR=> bError, 
	ERRID=> nErrorId );

END_FUNCTION_BLOCK

// CNC/3 Control/HLI3_GetChannelActiveG
FUNCTION_BLOCK HLI3_GetChannelActiveG
VAR_INPUT
	bExec:	   BOOL;			// riding edge to start read
	nChanIdx: INT;    			// zero based channel index	
END_VAR
VAR_OUTPUT
	ActiveG : ARRAY[0..39] OF INT;
	bBusy: BOOL;
	bError: BOOL;
	nErrorID: UDINT;
END_VAR
VAR
	fbAdsRead: ADSREAD;
END_VAR

(* ========================================================= *)
(*    FUN: HLI3_GetChannelActiveG                   		 *)
(* --------------------------------------------------------- *)
(*   Desc: Gets the channel specific active G functions      *)
(*															 *)
(* Return: Array[0..39] filled with the G information (<> -1)*)
(* Author: MiB                                               *)
(*   Date: 12.01.2016                                        *)
(*   Rev.: 1.0                                               *)
(* ========================================================= *)

fbAdsRead(
	NETID:= '' , 
	PORT:= 553, 
	IDXGRP:= 16#20100 + INT_TO_UDINT(nChanIdx) + 1, 
	IDXOFFS:= 16#3C , 
	LEN:= SIZEOF(ActiveG) , 
	DESTADDR:= ADR(ActiveG),
	READ:= bExec, 
	TMOUT:= , 
	BUSY=> bBusy, 
	ERR=> bError, 
	ERRID=> nErrorId );

END_FUNCTION_BLOCK

// CNC/3 Control/HLI3_GetChannelMessage
FUNCTION_BLOCK HLI3_GetChannelMessage
VAR_INPUT
	/// Number of channel 
	nChanIdx: INT;
	bExecute: BOOL := FALSE;
	bShowDlg: BOOL := FALSE;
END_VAR
VAR_OUTPUT
	strToPLC: STRING(HLI_MSG_CONTENT_STRL) := '';
	iMsgType: DWORD := 0;
END_VAR
VAR
	pChannel: POINTER TO HIGH_LEVEL_INTERFACE_CH;
	pMsgCU: POINTER TO MC_CONTROL_MSG_UNIT;
	pMsgToPLC: POINTER TO STRING(HLI_MSG_CONTENT_STRL);
END_VAR

(* ========================================================= *)
(*     FB: HLI_GetChannelMessage                             *)
(* --------------------------------------------------------- *)
(*   Desc: Get message from the CNC                          *)
(*   Author: MK, MiB                                         *)
(*   Date: 20.11.2012                                        *)
(*   Last:                                                   *)
(*   Rev.: 1.01                                              *)
(* ========================================================= *)

IF NOT HLI3_CheckChannelValid(nChannel := nChanIdx) THEN
	RETURN;
END_IF


(* Get pointer to data of a specific channel at the HLI *)
pChannel := gpCh[nChanIdx];

(* Control unit at the HLI that handles channel specific messages *)
pMsgCU := ADR(pChannel^.msg_mc_control);

IF bExecute = TRUE THEN
	(* Is the complete message in the control unit? *)
	IF pMsgCU^.request_semaphor_rw = TRUE
	THEN
		(* Pointer to content of the message sent to the PLC *)
		pMsgToPLC := ADR(pMsgCU^.request_r.inhalt);

		(* Get the message from the control unit *)
		strToPLC := pMsgToPLC^;

   	    CNCSystem.Channel[nChanIdx].Message := strToPLC;

		(* Get the message type *)
		iMsgType := pMsgCU^.request_r.typ;

		(* Pop up dialog with the message send to the PLC *)
		IF bShowDlg THEN
			ADSLOGSTR( msgCtrlMask := ADSLOG_MSGTYPE_MSGBOX OR ADSLOG_MSGTYPE_LOG,
			           msgFmtStr   := 'Message sent to PLC via HLI:%s',
			           strArg      := strToPLC);
		END_IF

		(* Acknowledge that you got the message *)
		pChannel^.msg_mc_control.request_semaphor_rw  := FALSE;
	END_IF;
END_IF;

END_FUNCTION_BLOCK

// CNC/3 Control/HLI3_GetFeedholdState
FUNCTION HLI3_GetFeedholdState : BOOL
VAR_INPUT
	/// Number of channel 
	nChanIdx: INT;
END_VAR


IF NOT HLI3_CheckChannelValid(nChannel := nChanIdx) THEN
	RETURN;
END_IF
HLI3_GetFeedholdState:=gpCh[nChanIdx]^.bahn_mc_control.feedhold.state_r;

END_FUNCTION

// CNC/3 Control/HLI3_GetIpoState
FUNCTION HLI3_GetIpoState : BOOL
VAR_INPUT
	nChanIdx: INT;
END_VAR



IF NOT HLI3_CheckChannelValid(nChannel := nChanIdx) THEN
	RETURN;
END_IF

HLI3_GetIpoState:=gpCh[nChanIdx]^.bahn_state.interpolation_active_r;

END_FUNCTION

// CNC/3 Control/HLI3_SetAxisGantryOn
FUNCTION HLI3_SetAxisGantryOn : BOOL
VAR_INPUT
	nHliAxisIdx: INT;
	bEnable: BOOL;
END_VAR

(****************************************************************************************)
(* POU:		HLI_SetAxisGantryOn                      									*)
(* Type:	Function																	*)
(* Author: 	HR																			*)
(* Date: 	11/01/24																	*)
(* Rev.: 	1.0																			*)
(* ------------------------------------------------------------------------------------ *)
(* Desc:	Enables the axis specific control unit for driving out the gantry			*)
(*			difference. The actual movement is triggered by the input 'bEnable'.		*)
(*			The current axis has to be a gantry slave. That means:						*)
(*				+ It is not attached to a channel										*)
(*				+ kenngr.achs_mode		0x2000n		(where n specifies the axis type)	*)
(*				+ kenngr.gantry_ax_nr	1			(e. g. axis no. of gantry master)	*)
(*				+ kenngr.gantry_offset  10000		(e. g. difference to be driven out)	*)
(*				+ kenngr.gantry_vb_korr	20000		(e. g. velocity for driving out)	*)
(****************************************************************************************)

(* Check specified logical axis no first *)
IF NOT HLI3_CheckAxisValid(nHliAxisIdx := nHliAxisIdx) THEN
	HLI3_SetAxisGantryOn := FALSE;
	RETURN;
END_IF

gpAx[nHliAxisIdx]^.lr_mc_control.gantry_on.enable_w	:= TRUE;
gpAx[nHliAxisIdx]^.lr_mc_control.gantry_on.command_w	:= bEnable;
HLI3_SetAxisGantryOn	:= TRUE;

END_FUNCTION

// CNC/3 Control/HLI3_SetAxisReferencePosition
FUNCTION HLI3_SetAxisReferencePosition : BOOL
VAR_INPUT
	bSetRefpos: BOOL;
	nHliAxisIdx: INT;
END_VAR

(* ========================================================= *)
(*    FUN: HLI_SetAxisReferenceposition                      *)
(* --------------------------------------------------------- *)
(*   Desc:                                                   *)
(* Author: HR                                                *)
(*   Date: 09.11.2010                                        *)
(*   Rev.: 1.0                                               *)
(* ========================================================= *)
HLI3_SetAxisReferencePosition := FALSE;

IF NOT HLI3_CheckAxisValid(nHliAxisIdx := nHliAxisIdx) THEN	
	RETURN;
END_IF

(* set reference position *)
gpAx[nHliAxisIdx]^.lr_mc_control.set_reference_position.command_w := bSetRefpos;
HLI3_SetAxisReferencePosition := TRUE;

END_FUNCTION

// CNC/3 Control/HLI3_SetAxisSpindleStopAtProgramEnd
FUNCTION_BLOCK HLI3_SetAxisSpindleStopAtProgramEnd
VAR_INPUT
	bExecute: BOOL;
	bSpindelStopAtProgramEnd: BOOL;
	nHliAxisIdx: INT;
END_VAR
VAR_OUTPUT
	bBusy: BOOL;
END_VAR
VAR
	/// Index of axis specific HLI area 
	nHliAxIfcIdx: INT;
	nState: INT;
	fbRTrigExecute: R_TRIG;
END_VAR

(****************************************************************************************)
(* POU:		HLI_SetAxisSpindleStopAtProgramEnd                      					*)
(* Type:		FB																		*)
(* Author: 	HR                                              							*)
(* Date: 	24.01.11																	*)
(* Rev.: 	1.0                                               							*)
(* ------------------------------------------------------------------------------------ *)
(* Desc:	Check wether the axis specified by input 'nLogAxisNo' is a spindle and 		*)
(*			(re-) sets (depending on the state of input 'bSpindelStopAtProgramEnd') 	*)
(*			the spindle stop feature on the HLI.										*)
(****************************************************************************************)

(****************************************************************************************)
(*								Check logical axis no									*)
(****************************************************************************************)
IF NOT HLI3_CheckAxisValid(nHliAxisIdx := nHliAxisIdx) THEN	
	RETURN;
END_IF
(****************************************************************************************)
(*									Build trigger										*)
(****************************************************************************************)
fbRTrigExecute
	(CLK := bExecute);

(****************************************************************************************)
(*								   (Re-)set sequence									*)
(****************************************************************************************)
CASE nState OF
 (* ----------------------------------------------------------------------------------- *)
 0: (* INIT STATE  *)
  	bBusy			:= FALSE;

	IF fbRTrigExecute.Q THEN
		bBusy		:= TRUE;
		nState		:= 10;
	END_IF

 (* ----------------------------------------------------------------------------------- *)
 10: (* ENABLE THE CONTROL UNIT IF THE AXIS IS A SPINDLE *)

	IF gpAx[nHliAxisIdx]^.ipo_state.spindle_axis_r THEN
		gpAx[nHliAxisIdx]^.ipo_mc_control.spdl_stop_at_prog_end.enable_w := TRUE;
		nState 		:= 20;
	ELSE
		nState 		:= 0;
	END_IF

 (* ---------------------------------------------------------------------------------- *)
 20: (* (RE-) SET SPINDLE STOP FUNCTION *)
	gpAx[nHliAxisIdx]^.ipo_mc_control.spdl_stop_at_prog_end.command_w := bSpindelStopAtProgramEnd;
	nState 			:= 0;
END_CASE

END_FUNCTION_BLOCK

// CNC/3 Control/HLI3_SetAxisTrackingOperation
FUNCTION HLI3_SetAxisTrackingOperation : BOOL
VAR_INPUT
	nHliAxisIdx: INT;
	bPLCAxisEnable: BOOL;
END_VAR

(* ========================================================= *)
(*    FUN: HLI_SetAxisTrackingOperation                      *)
(* --------------------------------------------------------- *)
(*   Desc:                                                   *)
(*   Author: TV                                              *)
(*   Date: 15.09.2006                                        *)
(*   Rev.: 1.0                                               *)
(*         1.1 13.08.2013 Nachführbetrieb nicht bei Achsfehler einschalten *)
(* ========================================================= *)

IF NOT HLI3_CheckAxisValid(nHliAxisIdx := nHliAxisIdx) THEN	
	HLI3_SetAxisTrackingOperation := FALSE;
	RETURN;
END_IF

(* tracking operation (follow up) on / off *)
IF NOT bPLCAxisEnable THEN
	gpAx[nHliAxisIdx]^.lr_mc_control.follow_up.command_w := TRUE;
		HLI3_SetAxisTrackingOperation := TRUE;
ELSE
	gpAx[nHliAxisIdx]^.lr_mc_control.follow_up.command_w := FALSE;
		HLI3_SetAxisTrackingOperation := FALSE;
END_IF

END_FUNCTION

// CNC/4 MHT-Function/HLI3_FastMFunctionHandler
FUNCTION_BLOCK HLI3_FastMFunctionHandler
VAR_INPUT
	bForceOff			: BOOL;													(* Forces all bytes in the output array to be 00 and therefore to switch off the digital output *) 
	bReset				: BOOL;													(* Resets the digital output *)
	nFunctionNoOn		: UINT;													(* Specifies the M function number for switching the digital output on *) 
	nDelayOn			: DINT;													(* Specifies a delay time in [µs] for switching on the digital output *)
	nFunctionNoOff		: UINT;													(* Specifies the M function number for switching the digital output off *)
	nDelayOff			: DINT;													(* Specifies a delay time in [µs] for switching off the digital output *)
	stData				: ST_FastMFunctionData;									(* Structure provided by an instance of HLI3_FastMFunctionProvider *)
END_VAR
VAR_OUTPUT
	abyOutput			: ARRAY[0..MAX_FAST_M_FUNC_OUTPUT_IDX] OF BYTE;		(* Output array for a digital oversampling output terminal EL2262 *)  
END_VAR
VAR
	bSwitchOn			: BOOL;
	nSwitchOnOffset		: DINT;
	bSwitchOff			: BOOL;
	nSwitchOffOffset	: DINT;
	bStateChanged		: BOOL;
	bFirstCycle			: BOOL := TRUE;
	byStaticValue		: BYTE;
	byBitmask			: BYTE;
	nBits				: DINT;
	nBytes				: DINT;
	nLoop				: UINT;
	nQueuedCount		: UINT;
	
	eLastState			: E_FastMFunctionState := E_FastMFunctionState.OFF;
	stDequeued			: ST_FastMFunctionBufferItem;
	astQueue			: ARRAY[0..MAX_FAST_M_FUNC_QUEUE_IDX] OF ST_FastMFunctionBufferItem;
	
	fbRtrigReset		: Tc2_Standard.R_TRIG;
	CYCLE_TIME			: UINT := 1000;
END_VAR

(****************************************************************************************)
(* POU:		HLI3_FastMFunctionHandler                     								*)
(* Type:	FB																			*)
(* Author: 	RCH		                                             						*)
(* Date: 	14/10/29																	*)
(* Rev.: 	1.0                                               							*)
(* ------------------------------------------------------------------------------------ *)
(* Desc.:	Function block for handling the oversampled output on an EL2262. The 		*)
(*			output state will be derived from the occurance of two CNC M functions, 	*)
(*			which have to be configured with output method MOS_TS and which have to be	*)
(*			preprocessed by an instance of the HLI3_FastMFunctionProvider function 		*)
(*			block. The switch ON/OFF times can be delayed seperately.					*)					
(*																						*)
(*			THIS FB HAS TO BE CALLED CYCLICALLY IN A 1MS TASK AND THE EL2262 HAS TO 	*)
(*			FEATURE AN OVERSAMPLING FACTOR OF 1000 (125 BYTE) ==> 1µs == 1 bit!!!		*)
(* ------------------------------------------------------------------------------------ *)
(* Rev.:	1.1																			*)
(* Date:	15/05/05								                                   	*)
(* Author:	RCH																		 	*)
(* Desc.:	Fixed issues occured if more than 1 MOS_TS M function was programmed in a   *)
(*			single G-Code block.														*)
(* ------------------------------------------------------------------------------------ *)
(* Rev.:	<Enter revision number here>												*)
(* Date:	<Enter revision data here>				                                   	*)
(* Author:	<Enter author´s shortcut here>											 	*)
(* Desc.:	<Enter description here>													*)
(****************************************************************************************)

(****************************************************************************************)
(*	  						  Refresh buffered switch times 							*)
(****************************************************************************************)
THIS^.RefreshQueue(CYCLE_TIME);

(****************************************************************************************)
(*	  							 	  Reset output										*)
(****************************************************************************************)
fbRtrigReset(CLK:= bReset);

IF fbRtrigReset.Q THEN
	THIS^.ClearQueue();
	bStateChanged				:= TRUE;
	eLastState					:= E_FastMFunctionState.OFF;
END_IF

(****************************************************************************************)
(*	  					    Search for new switch on/off events 						*)
(****************************************************************************************)
bSwitchOn						:= FALSE;
nSwitchOnOffset					:= 0;
bSwitchOff						:= FALSE;
nSwitchOffOffset				:= 0;
nLoop							:= 0;

IF (stData.nFunctionCount > 0) AND (stData.bDataValid) THEN
	REPEAT
		IF (stData.astItem[nLoop].nFunctionNo = nFunctionNoOn) THEN
			bSwitchOn			:= TRUE;
			nSwitchOnOffset		:= stData.astItem[nLoop].nOffset;
		ELSIF (stData.astItem[nLoop].nFunctionNo = nFunctionNoOff) THEN
			bSwitchOff			:= TRUE;
			nSwitchOffOffset	:= stData.astItem[nLoop].nOffset;
		END_IF
	
		nLoop					:= nLoop + 1;
		
		UNTIL ((bSwitchOn AND bSwitchOff) OR (nLoop >= stData.nFunctionCount))
	END_REPEAT	
END_IF

(****************************************************************************************)
(*	  		Buffer found switch on/off events with correspondent switch times			*)
(****************************************************************************************)
IF bSwitchOn AND bSwitchOff THEN
	(* In case switch on and off events have been transmitted within the same cycle, 	*)
	(* order them according to their switch times!										*)
	IF ((nSwitchOnOffset + nDelayOn) < (nSwitchOffOffset + nDelayOff)) THEN
		THIS^.Enqueue(E_FastMFunctionState.ON, nSwitchOnOffset + nDelayOn);
		THIS^.Enqueue(E_FastMFunctionState.OFF, nSwitchOffOffset + nDelayOff); 
	ELSE
		THIS^.Enqueue(E_FastMFunctionState.OFF, nSwitchOffOffset + nDelayOff);
		THIS^.Enqueue(E_FastMFunctionState.ON, nSwitchOnOffset + nDelayOn);
	END_IF
ELSIF bSwitchOn THEN
	THIS^.Enqueue(E_FastMFunctionState.ON, nSwitchOnOffset + nDelayOn);
ELSIF bSwitchOff THEN
	THIS^.Enqueue(E_FastMFunctionState.OFF, nSwitchOffOffset + nDelayOff);
END_IF

(****************************************************************************************)
(*	  				  Set output array according to latest switch state					*)
(****************************************************************************************)
IF bStateChanged OR bFirstCycle THEN
	bStateChanged				:= FALSE;

	IF (eLastState = E_FastMFunctionState.OFF) THEN
		byStaticValue			:= 16#00;
	ELSIF (eLastState = E_FastMFunctionState.ON) THEN
		byStaticValue			:= 16#FF;
	END_IF
	
	Tc2_System.MEMSET(ADR(abyOutput[0]), byStaticValue, SIZEOF(abyOutput));
END_IF

(****************************************************************************************)
(*	  					  Dequeue switch events from the buffer							*)
(****************************************************************************************)
WHILE THIS^.DequeuingRequired DO
	stDequeued					:= THIS^.Dequeue();
	nBits 						:= stDequeued.nSwitchTime MOD 8;
	nBytes 						:= stDequeued.nSwitchTime / 8;
	bStateChanged				:= TRUE;
	IF (stDequeued.nSwitchTime < 0) OR (stDequeued.nSwitchTime > 1000) THEN
		;
	ELSE
		IF ((stDequeued.eState = E_FastMFunctionState.ON) AND (eLastState = E_FastMFunctionState.OFF)) THEN
			byBitmask			:= SHL(BYTE#255, nBits);
			abyOutput[nBytes]	:= abyOutput[nBytes] OR byBitmask;
			eLastState			:= E_FastMFunctionState.ON;
			Tc2_System.MEMSET(ADR(abyOutput[nBytes + 1]), 16#FF, MAX_FAST_M_FUNC_OUTPUT_IDX - nBytes);
		ELSIF ((stDequeued.eState = E_FastMFunctionState.OFF) AND (eLastState = E_FastMFunctionState.ON)) THEN
			byBitmask			:= SHR(BYTE#255, 8 - nBits);
			abyOutput[nBytes]	:= abyOutput[nBytes] AND byBitmask;
			eLastState			:= E_FastMFunctionState.OFF;
			Tc2_System.MEMSET(ADR(abyOutput[nBytes + 1]), 16#00, MAX_FAST_M_FUNC_OUTPUT_IDX - nBytes);
		END_IF
	END_IF
END_WHILE

(****************************************************************************************)
(*	  							   Reset first cycle indicator							*)
(****************************************************************************************)
bFirstCycle						:= FALSE;

METHOD ClearQueue
Tc2_System.MEMSET(ADR(astQueue), 16#00, SIZEOF(astQueue));
nQueuedCount := 0;
END_METHOD

METHOD Dequeue : ST_FastMFunctionBufferItem
VAR
	stReturn	: ST_FastMFunctionBufferItem;
END_VAR
IF (nQueuedCount > 0) THEN
	stReturn		:=	astQueue[0]; 
	Tc2_System.MEMMOVE(ADR(astQueue[0]), ADR(astQueue[1]), SIZEOF(astQueue) - SIZEOF(stReturn));
	
	nQueuedCount	:= nQueuedCount - 1;
	Dequeue			:= stReturn;
END_IF
END_METHOD

PROPERTY DequeuingRequired : BOOL
GET
DequeuingRequired	:= (nQueuedCount > 0) AND 
					   (astQueue[0].eState <> E_FastMFunctionState.EMPTY) AND
					   (astQueue[0].nSwitchTime < CYCLE_TIME);
END_GET
END_PROPERTY

METHOD Enqueue
VAR_INPUT
	eState			: E_FastMFunctionState;
	nSwitchTime		: DINT;
END_VAR
IF (nQueuedCount <= MAX_FAST_M_FUNC_OUTPUT_IDX) THEN
	astQueue[nQueuedCount].eState		:= eState;
	astQueue[nQueuedCount].nSwitchTime	:= nSwitchTime;
	nQueuedCount						:= nQueuedCount + 1;
END_IF
END_METHOD

METHOD RefreshQueue
VAR_INPUT
	nCycleTime: UINT;
END_VAR
IF (nQueuedCount > 0) THEN
	FOR nLoop := 0 TO (nQueuedCount - 1) DO
		astQueue[nLoop].nSwitchTime	:= astQueue[nLoop].nSwitchTime - nCycleTime;
	END_FOR
END_IF
END_METHOD

END_FUNCTION_BLOCK

// CNC/4 MHT-Function/HLI3_FastMFunctionProvider
FUNCTION_BLOCK HLI3_FastMFunctionProvider
VAR_INPUT
	nHliChanIdx				: UINT;													(* HLI channel index of the channel to check for new M functions *)
	anMFunctionNo			: ARRAY[0..MAX_FAST_M_FUNC_ITEM_IDX] OF UINT;			(* List of M functions munbers to handle *)
END_VAR
VAR_OUTPUT
	stData					: ST_FastMFunctionData;									(* Output structure containing informatione about the handled M functions and their execution offsets *)
	bUnknownChannelIndex	: BOOL;													(* TRUE if the given nHliChanIdx is unknown *)
END_VAR
VAR
	bExitAll				: BOOL;
	bFirstCycle				: BOOL := TRUE;
	byTaskIndex				: BYTE;
	nConfiguredFunctions	: UINT;
	nFunctionCount			: UINT;
	nLoop1					: UINT;
	nLoop2					: UINT;
	anMFunctionNoOld		: ARRAY[0..MAX_FAST_M_FUNC_ITEM_IDX] OF UINT;
	pChan					: POINTER TO HIGH_LEVEL_INTERFACE_CH;
	pData					: POINTER TO ST_FastMFunctionItem;
	pTechno					: POINTER TO Techno_Unit_Ch;
	pMHTechno				: POINTER TO HLI_M_H_Prozess;
	
	fbGetTaskIndex			: Tc2_System.GETCURTASKINDEX;
END_VAR

(****************************************************************************************)
(* POU:		HLI3_FastMFunctionProvider                     								*)
(* Type:	FB																			*)
(* Author: 	RCH		                                             						*)
(* Date: 	14/10/29																	*)
(* Rev.: 	1.0                                               							*)
(* ------------------------------------------------------------------------------------ *)
(* Desc.:	FB for handling CNC M functions contained in the input array				*)
(*			'anMFunctionNo'. These M functions have to be configured as MOS_TS. Their	*)
(*			metadata will be copied into the output structure 'stData' to be processed	*)
(*			by instances of the FB HLI3_FastMFunctionHandler!							*)				
(*																						*)
(*			THIS FB HAS TO BE CALLED CYCLICALLY IN A 1MS TASK!!!						*)
(* ------------------------------------------------------------------------------------ *)
(* Rev.:	1.1																			*)
(* Date:	15/05/05								                                   	*)
(* Author:	RCH																		 	*)
(* Desc.:	Fixed issues occured if more than 1 MOS_TS M function was programmed in a   *)
(*			single G-Code block.														*)
(* ------------------------------------------------------------------------------------ *)
(* Rev.:	<Enter revision number here>												*)
(* Date:	<Enter revision data here>				                                   	*)
(* Author:	<Enter author´s shortcut here>											 	*)
(* Desc.:	<Enter description here>													*)
(****************************************************************************************)

(****************************************************************************************)
(*	  Read current (PLC) task id and check whether the cycle time has been exceeded		*)
(****************************************************************************************)
IF bFirstCycle THEN
	fbGetTaskIndex
		(index				=> byTaskIndex);
END_IF

(****************************************************************************************)
(*								Initialize output structure								*)
(****************************************************************************************)
Tc2_System.MEMSET(ADR(stData), 16#00, SIZEOF(stData));

stData.bCycleTimeExceeded	:= TwinCAT_SystemInfoVarList._TaskInfo[byTaskIndex].CycleTimeExceeded;
stData.bDataValid			:= FALSE;
stData.nFunctionCount		:= 0;	

(****************************************************************************************)
(*	  					  Check existence of the given channel index					*)
(****************************************************************************************)
IF NOT HLI3_CheckChannelValid(nChannel := nHliChanIdx) THEN
	bUnknownChannelIndex	:=	TRUE; 
	RETURN;
ELSE
	bUnknownChannelIndex	:=	FALSE;
END_IF

(****************************************************************************************)
(*	  				  Determine the number of configured M functions					*)
(****************************************************************************************)
IF (Tc2_System.MEMCMP(ADR(anMFunctionNo), ADR(anMFunctionNoOld), SIZEOF(anMFunctionNo)) <> 0) THEN
	anMFunctionNoOld				:= anMFunctionNo;
	nConfiguredFunctions			:= 0;
	
	FOR nLoop1 := 0 TO MAX_FAST_M_FUNC_ITEM_IDX DO
		IF (anMFunctionNoOld[nLoop1] > 0) THEN
			nConfiguredFunctions	:= nConfiguredFunctions + 1;
		END_IF
	END_FOR
END_IF

(****************************************************************************************)
(*	  					  	Check occurances of M functions								*)
(****************************************************************************************)
stData.bDataValid					:= TRUE;
bFirstCycle							:= FALSE;

IF (gpCh[nHliChanIdx]^.used_units_std_sync_r = 0) THEN
	RETURN;
END_IF

pChan								:= gpCh[nHliChanIdx];
nFunctionCount						:= 0;
nLoop1 								:= 0;

FOR nLoop1 := 0 TO INT_TO_UINT(HLI_TU_CH_STD_SYNC_MAXIDX) DO
	IF pChan^.techno_unit_std_sync[nLoop1].please_rw AND (pChan^.techno_unit_std_sync[nLoop1].fkt_ctrl_r = Tc2_CncHli.HLI_INTF_M_FKT) THEN
		pTechno						:= ADR(pChan^.techno_unit_std_sync[nLoop1]);
		pMHTechno					:= ADR(pTechno^.attribut_r);	
		
		(* Check whether this FB has to handle the current M function *)
		FOR nLoop2 := 0 TO (nConfiguredFunctions - 1) DO
			IF (pMHTechno^.nr = anMFunctionNo[nLoop2]) THEN
				pData				:= ADR(stData.astItem[nFunctionCount]);
				pData^.nFunctionNo	:= anMFunctionNo[nLoop2];
				pData^.nOffset		:= pMHTechno^.zeit;
				pData^.nCycleCount	:= TwinCAT_SystemInfoVarList._TaskInfo[byTaskIndex].CycleCount;
				
				nFunctionCount		:= nFunctionCount + 1;
				
				pTechno^.please_rw	:= FALSE;
				pTechno^.done_w		:= TRUE;		
				EXIT;	
			END_IF					
		END_FOR
		
		IF (nFunctionCount >= nConfiguredFunctions) THEN
			EXIT;
		END_IF
	ELSIF NOT pChan^.techno_unit_std_sync[nLoop1].please_rw THEN
		EXIT;
	END_IF	
END_FOR

stData.nFunctionCount				:= nFunctionCount;

END_FUNCTION_BLOCK

// CNC/4 MHT-Function/HLI3_QuitAxisMFunction
FUNCTION HLI3_QuitAxisMFunction : BOOL
VAR_INPUT
	/// Number of axis 
	nHliAxisIdx: INT;
END_VAR
VAR
	/// Data of a M/H techno unit 
	pMHProcess: POINTER TO HLI_M_H_PROZESS;
	/// Data of a spindle unit 
	pSProcess: POINTER TO HLI_S_PROZESS;
	/// Data of a techno unit 
	pTProcess: POINTER TO HLI_T_PROZESS;
	/// local pointer to Data of actual Axis 
	pAxisData: POINTER TO HIGH_LEVEL_INTERFACE_AX;
	/// local pointer to actual techno unit 
	pActTechnoUnit: POINTER TO TECHNO_UNIT_AX;
	/// loop variable 
	idx: UINT;
	/// Index of axis specific technology function at HLI 
	nTechFctMaxIdx: UINT;
	/// basis id of a tool 
	nToolBasicId: UDINT;
	/// spindle movement command 
	SpdlMoveCmd: UINT;
	/// SpindleRevolution 
	Revolution: UDINT;
	/// SpindleRevolution 
	pRevolution: POINTER TO UDINT;
	/// Number of M-function 
	FuncNr: UDINT;
END_VAR

(* ========================================================= *)
(*    FUN: HLI_QuitAxisMFunction                             *)
(* --------------------------------------------------------- *)
(*   Desc:                                                   *)
(* Author: MK                                                *)
(*   Rev.: 1.1                                               *)
(*   Date: 18.07.2002                                        *)
(*       : 08.04.2005                                        *)
(* ========================================================= *)

HLI3_QuitAxisMFunction := FALSE;
IF NOT (HLI3_CheckAxisValid(nHliAxisIdx := nHliAxisIdx)) THEN
	RETURN;
END_IF


(* get pointer to Axis data *)
pAxisData := gpAx[nHliAxisIdx];

(* test if there are open synchronisations  *)
IF pAxisData^.used_units_std_sync_r > 0 THEN

	nTechFctMaxIdx := pAxisData^.used_units_std_sync_r - 1;

	FOR idx := 0 TO nTechFctMaxIdx DO
	
		(* get pointer to actual techno unit *)
		pActTechnoUnit := ADR(pAxisData^.techno_unit_std_sync[idx]);
	
		(* test if this M-function has to be acknowledged *)
		IF pActTechnoUnit^.please_rw = TRUE AND				(* request from CNC *)
			pActTechnoUnit^.done_w = FALSE					(* not acknowledged *)
		THEN
	
			IF pActTechnoUnit^.fkt_ctrl_r = HLI_INTF_M_FKT THEN
				(* Example: read number of M-function *)
				pMHProcess := ADR(pActTechnoUnit^.attribut_r.data[0]);
				FuncNr := pMHProcess^.nr;
				//ADSLOG(strMsg:='Axis acknowledge of M-function: %d', nDINT:=UDINT_TO_DINT(FuncNr), strArg:='');
			ELSE
				IF pActTechnoUnit^.fkt_ctrl_r = HLI_INTF_SPINDEL THEN (* spindle-fuction *)
					pSProcess := ADR(pActTechnoUnit^.attribut_r.data[0]);
	
					(* Example: read revolution of S-function *)
					Revolution := DINT_TO_UINT(pSProcess^.rev);
					//ADSLOG(strMsg:='Spindle S-function: %d', nDINT:=UDINT_TO_DINT(Revolution), strArg:='');
	
					(* Example: read number of S-function *)
					SpdlMoveCmd := pSProcess^.move_cmd;
					//ADSLOG(strMsg:='Spindle acknowledge of M-function: %d', nDINT:=SpdlMoveCmd, strArg:='');
				ELSE
					ADSLOGDINT( msgCtrlMask :=    ADSLOG_MSGTYPE_MSGBOX
					                           OR ADSLOG_MSGTYPE_LOG,
								msgFmtStr   := 'Axis acknowledge unknown type: %d',
								dintArg     := pActTechnoUnit^.fkt_ctrl_r);
				END_IF
			END_IF
	
			(* acknowledge this M-function *)
			pActTechnoUnit^.please_rw := FALSE;
			pActTechnoUnit^.done_w := TRUE;
	
			HLI3_QuitAxisMFunction := TRUE;
		END_IF
	END_FOR

END_IF

END_FUNCTION

// CNC/5 Variables/FB_ReadCNCVariables
FUNCTION_BLOCK FB_ReadCNCVariables
VAR_INPUT
	bEnable		:	BOOL ;	(* B *)
	nChanIdx	:   INT;
	eVariablesType : E_CNCVariablesType;
	tIntervall	:   TIME;
END_VAR

VAR_OUTPUT
	Done			:	BOOL;	(* B *)
	Busy			: 	BOOL;	(* E *)	
	Error			:	BOOL;	(* B *)
	ErrorID			:	UDINT;	(* E *) 
END_VAR

VAR_IN_OUT
	 stCNCVariablesViewer_Data : ARRAY[0..MAX_CNC_VAR_LIST_IDX] OF ST_CNCVariablesViewer_Data;
END_VAR

VAR	
	fbTrigger :	R_TRIG;
	fbReadNumber: ADSREAD;
	nParameterNumber : DINT;
		
	fbReadWrite: ADSRDWRT;	
	strVarName : STRING(96);	
	fVarValue  : LREAL;    
 	nIndex     : UDINT;
	nListIndex : UDINT;	
	
	nState	: INT;
	fbTimer : TON;

	nReadLength 	   : UDINT;
	
 	IDXOffsNumber	   : UDINT;
	IDXOffsNamebyIndex : UDINT;
	IDXOffsValuebyIndex : UDINT;	
	stCNCVariablesViewer_Data_Temp : ARRAY[0..MAX_CNC_VAR_LIST_IDX] OF ST_CNCVariablesViewer_Data;
		
	nVEType 				: DINT;
	nVESize 	 			: UDINT;
    nVEMaxIndex1 		   	: UDINT; 
    nVEMaxIndex2 		   	: UDINT;
	strVEVarName 			: STRING(255);	
	strVEDisplayVarName		: STRING(255);
	arrVEDescriptionInput  	: ARRAY[0..259] OF BYTE;
	arrVEOutput 			: ARRAY[0..2047] OF BYTE;
			
	nVEArrayIndex       	: UDINT;
	nListIndexArrayStart	: UDINT; 	
	
	strValue            : STRING(799);
			
	dummyBoolean		: BOOL;
	dummySInt			: SINT;
	dummyUSInt			: USINT;
	dummyInt            : INT;
	dummyUInt			: UINT;
	dummyDInt           : DINT;
	dummyUDInt          : UDINT;
	dummyLReal          : LREAL;
	dummyString         : STRING;
	dummyLargeString    : STRING(799);  

	eVariablesTypeOld : E_CNCVariablesType;
	
END_VAR

VAR CONSTANT
	IDXOffsPNumber  : UDINT := 16#2;	
	IDXOffsVLNumber : UDINT := 16#3;
	IDXOffsVPNumber : UDINT := 16#4;
	IDXOffsVSNumber : UDINT := 16#5;
			
	IDXOffsPNamebyIndex : UDINT := 16#1B;
	IDXOffsVLNamebyIndex : UDINT := 16#1E;
	IDXOffsVPNamebyIndex : UDINT := 16#21;
	IDXOffsVSNamebyIndex : UDINT := 16#24;		
	
	IDXOffsPValuebyIndex : UDINT := 16#1D;
	IDXOffsVLValuebyIndex : UDINT := 16#20;
	IDXOffsVPValuebyIndex : UDINT := 16#23;
	IDXOffsVSValuebyIndex : UDINT := 16#26;
	IDXOffsVEValuebyName : UDINT := 16#2E;		
END_VAR

(****************************************************************************************)
(* POU:		ReadCNCVariables                     										*)
(* Type:	FB																			*)
(* Author: 	TV , MiB                                       								*)
(* Date: 	20.01.2016, 19.12.2016														*)
(* Rev.: 	1.0                                              							*)
(* Rev.: 	1.1 MiB VStrings support (up to 800byte)           							*)
(* ------------------------------------------------------------------------------------ *)
(* Desc:	Description																	*)
(****************************************************************************************)

(****************************************************************************************)
(*	FB reads in P, V.P, V.L., V.S., V.E. Parameter from the CNC Kernel via ADS		    *)
(****************************************************************************************)

IF (NOT HLI3_CheckChannelValid(nChannel := nChanIdx)) THEN	
	RETURN; (* A b b r u c h *)
END_IF

IF 	NOT bEnable OR 
	eVariablesType = E_CNCVariablesType.none  OR
	(gpCh[0]^.channel_mc_control.mode_and_state.state_r.mode = HLI_IMCM_MANUAL_MODE AND eVariablesType <> E_CNCVariablesType.VE) OR
	(gpCh[nChanIdx]^.channel_mc_control.mode_and_state.state_r.state <> HLI_IMCM_PROCESS_ACTIVE AND 
	gpCh[nChanIdx]^.channel_mc_control.mode_and_state.state_r.state <>  HLI_IMCM_PROCESS_HOLD AND eVariablesType <> E_CNCVariablesType.VE) 
		
	THEN
		Tc2_System.MEMSET(ADR(stCNCVariablesViewer_Data),0,SIZEOF(stCNCVariablesViewer_Data));
		fbTrigger(CLK:= FALSE);
		nState := 0;  
	ELSE
		fbTrigger(CLK:= TRUE);	
END_IF

IF fbTrigger.Q OR eVariablesTypeOld <> eVariablesType THEN		
	fbReadNumber(READ:= FALSE);
	fbReadWrite(WRTRD:= FALSE);
	nIndex 		:= 1;	
	nListIndex  := 0;
	nState 		:= 1;
	Error		:= FALSE;	(* B *)
	ErrorID		:= 0;		(* E *) 
END_IF

IF nState <> 0 THEN
	Busy := TRUE;
END_IF

CASE nState OF
	
0:
;  
1: 
	Error		:= FALSE;	(* B *)
	ErrorID		:= 0;	(* E *)

	eVariablesTypeOld :=  eVariablesType;
 
	Tc2_System.MEMSET(ADR(stCNCVariablesViewer_Data_Temp),0,SIZEOF(stCNCVariablesViewer_Data_Temp));
	
   	IF (eVariablesType = E_CNCVariablesType.P) THEN
	      IDXOffsNumber 	 	:= IDXOffsPNumber;
		  IDXOffsNamebyIndex 	:= IDXOffsPNamebyIndex;
		  IDXOffsValuebyIndex 	:= IDXOffsPValuebyIndex;
		  nReadLength			:= 8;			  
	ELSIF (eVariablesType = E_CNCVariablesType.VL) THEN
		 IDXOffsNumber 		 	:=  IDXOffsVLNumber;
		 IDXOffsNamebyIndex  	:= IDXOffsVLNameByIndex;
		 IDXOffsValuebyIndex 	:= IDXOffsVLValuebyIndex;
		 nReadLength			:= 8;
	ELSIF (eVariablesType = E_CNCVariablesType.VP) THEN
		 IDXOffsNumber 		 	:=  IDXOffsVPNumber;
		 IDXOffsNamebyIndex  	:= IDXOffsVPNameByIndex;
		 IDXOffsValuebyIndex 	:= IDXOffsVPValuebyIndex;
		 nReadLength			:= 8;
	ELSIF (eVariablesType = E_CNCVariablesType.VS) THEN
		 IDXOffsNumber 		 	:=  IDXOffsVSNumber;
		 IDXOffsNamebyIndex  	:= IDXOffsVSNameByIndex;
		 IDXOffsValuebyIndex 	:= IDXOffsVSValuebyIndex;
		 nReadLength			:= 8;	
   	END_IF
				
	
	IF (eVariablesType <> E_CNCVariablesType.VE) THEN
		fbReadNumber(
			NETID:= , 
			PORT:= 552, 
			IDXGRP:= 16#22300 + INT_TO_UDINT(nChanIdx)+1, 
			IDXOFFS:= IDXOffsNumber, 
			LEN:= 4, 
			DESTADDR:= ADR(nParameterNumber), 
			READ:= TRUE, 
		);
		
		IF NOT fbReadNumber.Busy THEN
			IF fbReadNumber.Err	THEN
				Error := fbReadNumber.ERR;
				ErrorID := fbReadNumber.ERRID;
				nState := 99;
			ELSE			
				nState := nState + 1;				
			END_IF
		END_IF
	ELSE
		nState := 20;
	END_IF

2:	// Read Variablen Name	
	IF nParameterNumber > 0 THEN 
		fbReadWrite(
		NETID:= , 
		PORT:= 552, 
		IDXGRP:= 16#22300 + INT_TO_UDINT(nChanIdx)+1, 
		IDXOFFS:= IDXOffsNamebyIndex, 
		WRITELEN:= 4, 
		READLEN:= 96, 
		SRCADDR:= ADR(nIndex), 
		DESTADDR:=ADR(strVarName), 
		WRTRD:= TRUE);
	
		IF NOT fbReadWrite.Busy THEN
			IF fbReadWrite.Err	THEN
				Error := fbReadWrite.ERR;
				ErrorID := fbReadWrite.ERRID;
				nState := 99;
			ELSE					
				fbReadWrite(WRTRD:= FALSE);	
				nState := 3;							
			END_IF
		END_IF
	
	ELSE	
		nState := 99;
	END_IF
	
	
3:	// Read Variablen Value	P V.L. V.P. V.S	
		fbReadWrite(
		NETID:= , 
		PORT:= 552, 
		IDXGRP:= 16#22300 + INT_TO_UDINT(nChanIdx)+1, 
		IDXOFFS:= IDXOffsValuebyIndex, 
		WRITELEN:= 4, 
		READLEN:= nReadLength, 
		SRCADDR:= ADR(nIndex), 
		DESTADDR:=ADR(fVarValue), 
		WRTRD:= TRUE);
	
		IF NOT fbReadWrite.Busy THEN
			IF fbReadWrite.Err	THEN
				Error := fbReadWrite.ERR;
				ErrorID := fbReadWrite.ERRID;
				nState := 99;
			ELSE
				stCNCVariablesViewer_Data_Temp[nListIndex].strName := strVarName;
				stCNCVariablesViewer_Data_Temp[nListIndex].strValue := LREAL_TO_STRING(fVarValue);		
				nListIndex := nListIndex+1;								
				nState := 4;
			END_IF
		END_IF		
		
		
4:  
	IF nIndex < DINT_TO_UDINT(nParameterNumber) AND (nListIndex <= MAX_CNC_VAR_LIST_IDX) THEN
		fbReadWrite(WRTRD:= FALSE);
		//nListIndex := nListIndex+1; 
		nIndex := nIndex + 1;
		nState := 2;
	ELSE
			fbTimer(IN:=FALSE);
			nState := 60;
	END_IF

20:    	// Read V.E. Variable element number
		arrVEDescriptionInput[0] := 86; // V
		arrVEDescriptionInput[1] := 46; //.
		arrVEDescriptionInput[2] := 69; //E
		
		fbReadWrite(
			NETID:= , 
			PORT:= 552, 
			IDXGRP:= 16#22300 + INT_TO_UDINT(nChanIdx)+1, 
			IDXOFFS:= 16#44, 
			WRITELEN:= 256, 
			READLEN:= 4, 
			SRCADDR:= ADR(arrVEDescriptionInput), 
			DESTADDR:=ADR(nParameterNumber), 
			WRTRD:= TRUE);

			IF NOT fbReadWrite.Busy THEN
				IF fbReadWrite.Err	THEN
					Error := fbReadWrite.ERR;
					ErrorID := fbReadWrite.ERRID;
					nState := 99;
				ELSE
					fbReadWrite(WRTRD:= FALSE);
					IF nParameterNumber > 0 THEN	
						nIndex := 0;		
						nListIndexArrayStart := 0;
						nVEArrayIndex := 0;			
						nState := 21;					
					ELSE			
						fbTimer(IN:=FALSE);
						nState := 60;			
					END_IF
				END_IF	
			END_IF			
			
21:		// Read V.E. Variable description by index
		MEMCPY(ADR(arrVEDescriptionInput),ADR(nIndex),SIZEOF(nIndex));
		arrVEDescriptionInput[4] := 86; // V
		arrVEDescriptionInput[5] := 46; //.
		arrVEDescriptionInput[6] := 69; //E
		
		fbReadWrite(
			NETID:= , 
			PORT:= 552, 
			IDXGRP:= 16#22300 + INT_TO_UDINT(nChanIdx)+1, 
			IDXOFFS:= 16#45, 
			WRITELEN:= 260, 
			READLEN:= 2048, 
			SRCADDR:= ADR(arrVEDescriptionInput), 
			DESTADDR:=ADR(arrVEOutput), 
			WRTRD:= TRUE);
	
		IF NOT fbReadWrite.Busy THEN
			IF fbReadWrite.Err	THEN
				Error := fbReadWrite.ERR;
				ErrorID := fbReadWrite.ERRID;
				nState := 99;
			ELSE
				fbReadWrite(WRTRD:= FALSE);
				
				//MEMCPY(ADR(nHandle),ADR(arrByte3),SIZEOF(nHandle));
				MEMCPY(ADR(nVEType),ADR(arrVEOutput)+4,SIZEOF(nVEType));
				// MEMCPY(ADR(nAccess),ADR(arrByte3)+4+4,SIZEOF(nAccess));
				MEMCPY(ADR(nVESize),ADR(arrVEOutput)+4+4+4,SIZEOF(nVESize));
				MEMCPY(ADR(nVEMaxIndex1),ADR(arrVEOutput)+4+4+4+4,SIZEOF(nVEMaxIndex1));
				IF nVEMaxIndex1 <> 0 THEN
					MEMCPY(ADR(nVEMaxIndex2),ADR(arrVEOutput)+4+4+4+4+4,SIZEOF(nVEMaxIndex2));
					MEMCPY(ADR(strVEVarName),ADR(arrVEOutput)+4+4+4+4+4+4,SIZEOF(strVEVarName));
				ELSE
					MEMCPY(ADR(strVEVarName),ADR(arrVEOutput)+4+4+4+4+4,SIZEOF(strVEVarName));
				END_IF
												
				IF nVEMaxIndex1 > 0 THEN
					nListIndexArrayStart := nListIndex;
					FOR nVEArrayIndex := 0 TO nVEMaxIndex2-1 DO						
						strVEDisplayVarName := CONCAT(strVEVarName,'[');
						strVEDisplayVarName := CONCAT(strVEDisplayVarName,UDINT_TO_STRING(nVEArrayIndex));
						strVEDisplayVarName := CONCAT(strVEDisplayVarName,']');			
						stCNCVariablesViewer_Data_Temp[nListIndex].strName := strVEDisplayVarName;
						IF (nListIndex < MAX_CNC_VAR_LIST_IDX) THEN
							nListIndex := nListIndex+1;
						ELSE
							EXIT;
						END_IF
							
					END_FOR	
					   nVEArrayIndex := 0;
					   nListIndex := nListIndexArrayStart;
					   nState := 25;											
				ELSE			
					nVEArrayIndex := 0;
					stCNCVariablesViewer_Data_Temp[nListIndex].strName := strVEVarName;						
					nState := 25;
				END_IF						
			END_IF
		END_IF	
		
25:		// Read Value By Name	
		IF nVEMaxIndex1 = 0 THEN			
			strVEVarName := stCNCVariablesViewer_Data_Temp[nListIndex].strName;
		ELSE
			strVEVarName := stCNCVariablesViewer_Data_Temp[nListIndex+nVEArrayIndex].strName ;
		END_IF		
							
		fbReadWrite(
		NETID:= , 
		PORT:= 552, 
		IDXGRP:= 16#22300 + INT_TO_UDINT(nChanIdx)+1, 
		IDXOFFS:= 16#48, 
		WRITELEN:= SIZEOF(strVEVarName), 
		READLEN:= 2048, 
		SRCADDR:= ADR(strVEVarName), 
		DESTADDR:=ADR(arrVEOutput), 
		WRTRD:= TRUE);
		
		IF NOT fbReadWrite.Busy THEN
			IF fbReadWrite.Err	THEN
				Error := fbReadWrite.ERR;
				ErrorID := fbReadWrite.ERRID;
				nState := 99;
			ELSE	
						
				IF nVEType = E_VEVariablesType.BOOLEAN THEN 
					MEMCPY(ADR(dummyBoolean),ADR(arrVEOutput),1);
					strValue := BOOL_TO_STRING(dummyBoolean);
				ELSIF nVEType = E_VEVariablesType.UNS08 THEN
					MEMCPY(ADR(dummyUSInt),ADR(arrVEOutput),1);
					strValue := USINT_TO_STRING(dummyUSInt);
				ELSIF nVEType = E_VEVariablesType.SGN08 THEN
					MEMCPY(ADR(dummySInt),ADR(arrVEOutput),1);
					strValue := SINT_TO_STRING(dummySInt);
				ELSIF nVEType = E_VEVariablesType.UNS16 THEN
					MEMCPY(ADR(dummyUInt),ADR(arrVEOutput),2);
					strValue := UINT_TO_STRING(dummyUInt);
				ELSIF nVEType = E_VEVariablesType.SGN16 THEN
					MEMCPY(ADR(dummyInt),ADR(arrVEOutput),2);
					strValue := INT_TO_STRING(dummyInt);
				ELSIF nVEType = E_VEVariablesType.UNS32 THEN
					MEMCPY(ADR(dummyUDInt),ADR(arrVEOutput),4);
					strValue := UDINT_TO_STRING(dummyUDInt);
				ELSIF nVEType = E_VEVariablesType.SGN32 THEN
					MEMCPY(ADR(dummyDInt),ADR(arrVEOutput),4);
					strValue := DINT_TO_STRING(dummyDInt);
				ELSIF nVEType = E_VEVariablesType.REAL64 THEN
					MEMCPY(ADR(dummyLReal),ADR(arrVEOutput),8);
					strValue := LREAL_TO_STRING(dummyLReal);						
				ELSIF nVEType = E_VEVariablesType.VESTRING THEN					 									
					MEMCPY(ADR(dummyLargeString),ADR(arrVEOutput),nVESize-1);
					strValue := dummyLargeString;
				ELSE
					nState := 99;
				END_IF				
				
				nState := 26;	
			END_IF
		END_IF	
		
26:
		stCNCVariablesViewer_Data_Temp[nListIndex+nVEArrayIndex].strValue := strValue;									
										
		IF nVEArrayIndex < nVEMaxIndex2-1 AND  nVEMaxIndex1 <> 0 THEN
			fbReadWrite(WRTRD:= FALSE);
			nVEArrayIndex := nVEArrayIndex +1;
			IF (nListIndex+nVEArrayIndex <= MAX_CNC_VAR_LIST_IDX) THEN
				nState := 25;
			ELSE
				nState := 60;
			END_IF
		ELSE
			IF (nListIndex <= MAX_CNC_VAR_LIST_IDX) THEN
				nListIndex := nListIndex+nVEArrayIndex +1;
				nState := 30;
			ELSE
				nState := 60;
			END_IF		
			
		END_IF
		
30:  
	IF nIndex < DINT_TO_UDINT(nParameterNumber-1) THEN
		fbReadWrite(WRTRD:= FALSE);		 
		nIndex := nIndex + 1;
		nState := 21;
	ELSE
		fbReadWrite(WRTRD:= FALSE);				
		fbTimer(IN:=FALSE);			
		nState := 60;
	END_IF

60:
	// Output
	Tc2_System.MEMCPY(ADR(stCNCVariablesViewer_Data),ADR(stCNCVariablesViewer_Data_Temp),SIZEOF(stCNCVariablesViewer_Data_Temp));
	fbTimer(IN:=TRUE , PT:=tIntervall);	
	IF fbTimer.Q THEN
		fbReadNumber(READ:= FALSE);
		fbReadWrite(WRTRD:= FALSE);
		nListIndex := 0;
		nIndex := 1;
		nState := 1;
	END_IF

99: // Error 
	nIndex := 1;
	nListIndex := 0;
	fbReadNumber(READ:= FALSE);
	fbReadWrite(WRTRD:= FALSE);
	fbTimer(IN:=FALSE);
	nState := 60;			
END_CASE

END_FUNCTION_BLOCK

// CNC/5 Variables/FB_ReadVxVar
FUNCTION_BLOCK FB_ReadVxVar
VAR_INPUT
	bExecute			: BOOL;   				(* rising edge commands start of FB *)
	strVarName 			: STRING(96); 			(* name of the Variable to read. Examples: V.G.WZ_AKT.L, V.A.MAX_POS.X, V.E.Template *)
	varType				: E_VxVariablesType; 	(* type of V.G. variable: use VariableViewer to get type of V.G. Variable *)
	nChanIdx			: INT;					(* zero based channel index *)	
	netId				: STRING := '';			(* NETID of target, local system if empty *)
END_VAR
VAR_OUTPUT
	bBusy			: 	BOOL;				(* fb is busy *)
	bError			:	BOOL;				(* error state *)
	nErrID			:	UDINT;				(* error id *)
	strError		: 	STRING(80);			(* error text *)
	strValue		: 	STRING(2048);		(* output value of V.x. Variable as string *)
	outBoolean		: BOOL;
	outSInt			: SINT;
	outUSInt		: USINT;
	outInt          : INT;
	outUInt			: UINT;
	outDInt         : DINT;
	outUDInt        : UDINT;
	outLReal        : LREAL;
	outString       : STRING(2048);
	
END_VAR
VAR
	fbReadWrite				: ADSRDWRT;	
	arrVxOutput 			: ARRAY[0..2047] OF BYTE;
	state 					: INT;
	exeTrig					: R_TRIG;
	
END_VAR

(**********************************************************************************************************
NAME...................:		FB_ReadVxVar	
Date...................:		2018.01.05
AUTHOR.................:		Michael Balsfulland (Beckhoff Automation GmbH & Co. KG)
VERSION................:		1.0
Description............:		read a V.G.or V.A.or V.E. variable via ADS 	
***********************************************************************************************************)

exeTrig(clk := bExecute);
	
IF (exeTrig.Q) THEN
	state := 10;
	bError := FALSE;
	nErrID := 0;
	strError := '';
	strValue := '';
	outBoolean := FALSE;
	outSInt := 0;
	outUSInt := 0;
	outInt := 0;
	outUInt := 0;
	outDInt := 0;
	outUDInt := 0;
	outLReal := 0.0;
	outString := '';
END_IF



CASE state OF
	0:  (* IDLE *)
		bBusy := FALSE;
	10:  (* Start *) 
		bBusy := TRUE;
		fbReadWrite( 	NETID:= netId , 
						PORT:= 552, 
						IDXGRP:= 16#22300 + INT_TO_UDINT(nChanIdx)+1, 
						IDXOFFS:= 16#48, 
						WRITELEN:= SIZEOF(strVarName), 
						READLEN:= 2048, 
						SRCADDR:= ADR(strVarName), 
						DESTADDR:=ADR(arrVxOutput), 
						WRTRD:= FALSE);
		state := state + 10;
		
	20:
		fbReadWrite(WRTRD := TRUE);
		IF NOT fbReadWrite.Busy THEN
			IF fbReadWrite.Err	THEN				
				nErrID := fbReadWrite.ERRID;
				strError := 'error in step 20 fb ADSRDWRT';
				state := 99;
			ELSE	
						
				IF varType = E_VxVariablesType.BOOLEAN THEN 
					MEMCPY(ADR(outBoolean),ADR(arrVxOutput),1);
					strValue := BOOL_TO_STRING(outBoolean);
				ELSIF varType = E_VxVariablesType.UNS08 THEN
					MEMCPY(ADR(outUSInt),ADR(arrVxOutput),1);
					strValue := USINT_TO_STRING(outUSInt);
				ELSIF varType = E_VxVariablesType.SGN08 THEN
					MEMCPY(ADR(outSInt),ADR(arrVxOutput),1);
					strValue := SINT_TO_STRING(outSInt);
				ELSIF varType = E_VxVariablesType.UNS16 THEN
					MEMCPY(ADR(outUInt),ADR(arrVxOutput),2);
					strValue := UINT_TO_STRING(outUInt);
				ELSIF varType = E_VxVariablesType.SGN16 THEN
					MEMCPY(ADR(outInt),ADR(arrVxOutput),2);
					strValue := INT_TO_STRING(outInt);
				ELSIF varType = E_VxVariablesType.UNS32 THEN
					MEMCPY(ADR(outUDInt),ADR(arrVxOutput),4);
					strValue := UDINT_TO_STRING(outUDInt);
				ELSIF varType = E_VxVariablesType.SGN32 THEN
					MEMCPY(ADR(outDInt),ADR(arrVxOutput),4);
					strValue := DINT_TO_STRING(outDInt);
				ELSIF varType = E_VxVariablesType.REAL64 THEN
					MEMCPY(ADR(outLReal),ADR(arrVxOutput),8);
					strValue := LREAL_TO_STRING(outLReal);
				ELSIF varType = E_VxVariablesType.VSTRING THEN					 									
					MEMCPY(ADR(outString),ADR(arrVxOutput) ,2048);
					strValue := outString;
						
				ELSE
					nErrID := 1;
					strError := 'error in step 20: varType not found';
					State := 99;
				END_IF				
				
				state := 30;
			END_IF
		END_IF	
		
	30: (* success *)
		state := 0;
			
	99: (* error *)
		bBusy := FALSE;
		bError := TRUE;
	
	
END_CASE

END_FUNCTION_BLOCK

// CNC/5 Variables/HLI3_GetVEChannelBooleanValue
FUNCTION HLI3_GetVEChannelBooleanValue : BOOL
VAR_INPUT
	/// HLI Channel Index
	nChanIdx: INT;
	/// Index of variable  range 1 ...     HLI_VE_VALUEMAX 
	nVEIndex: DINT;
	/// Array index. 0 if no array 
	nArrayIndex: DINT := 0;
	/// serves acess to the global variable array 
	bGlobal: BOOL;
END_VAR
VAR
	pVeData: POINTER TO VEData := 0;
	/// Size of the datatype of the returned value 
	iDatatypeSize: DINT;
	ptr: POINTER TO BOOL;
	ChIdx: UDINT;
	SizeField: DINT := 0;
END_VAR

(* ========================================================= *)
(*    FUN: GetVEChannelDINTValue                            *)
(* --------------------------------------------------------- *)
(*   Desc: Reads a V.E.Variable of Boolean                   *)
(* 	 Author: CL  / TV                                        *)
(*   Date: 16.05.2006                                        *)
(*   Last: 05.12.2013                                        *)
(*   Rev.: 1.3                                               *)
(* ========================================================= *)

IF  nVEIndex >= 0 AND
	nArrayIndex >= 0 THEN

	(* test if channel specific or global *)
	IF bGlobal = FALSE  THEN
		IF NOT HLI3_CheckChannelValid(nChannel := nChanIdx) THEN
			RETURN;
		END_IF
				
		pVeData := gpVECh[nChanIdx];
	ELSE
		pVeData := gpVEGlobal;
	END_IF

	IF pVeData <> 0 THEN
		IF pVeData <> 0 THEN
			iDatatypeSize := SIZEOF(ptr^);
                         	ptr := pVeData +  24  * nVEIndex + (iDatatypeSize * nArrayIndex);
                           HLI3_GetVEChannelBooleanValue := ptr^; (* successfully completed return *)
                END_IF
	END_IF
END_IF

END_FUNCTION

// CNC/5 Variables/HLI3_GetVEChannelDIntValue
FUNCTION HLI3_GetVEChannelDIntValue : DINT
VAR_INPUT
	/// HLI Channel Index 
	nChanIdx: INT;
	/// Index of variable  range 1 ...     HLI_VE_VALUEMAX 
	nVEIndex: DINT;
	/// Array index. 0 if no array 
	nArrayIndex: DINT := 0;
	/// serves acess to the global variable array 
	bGlobal: BOOL;
END_VAR
VAR
	pVeData: POINTER TO VEData := 0;
	/// Size of the datatype of the returned value 
	iDatatypeSize: DINT;
	ptr: POINTER TO DINT;
	ChIdx: UDINT;
	SizeField: DINT := 0;
END_VAR

